(* Visualisation VISU_1_ENGINE
rectangle at (20,550)-(331,601): text "%s"; shows INPUTS.sVisuTime
rectangle at (15,0)-(326,51): text "ENGINE"
rectangle at (45,420)-(226,441): text "Coolant Temperature:%.0f ºC"; shows RECV_J1939.FEEE.EngineCoolantTemperature
rectangle at (45,440)-(226,461): text "Fuel Temperature:	%.0f ºC"; shows RECV_J1939.FEEE.EngineFuelTemperature
rounded rectangle at (900,50)-(1021,101): alarm colour if MAIN.aSys_Enable[8]
rounded rectangle at (905,55)-(1016,96): text "ENABLE / ENGINE"; alarm colour if MAIN.aSys_Enable[8]; taps MAIN.SIEngineEnable.In
rounded rectangle at (905,505)-(1016,546): text "RETURN"; opens VISU_0_MAIN
rounded rectangle at (905,395)-(1016,436): text "CONFIG: / ENGINE"; opens VISU_CFG_ENGINE
rounded rectangle at (905,450)-(1016,491): text "CONFIG: / PROPULSION"; opens VISU_CFG_PROPULSION
rectangle at (0,0)-(1,1): text "{ExtendedElement},Visu\ElementDLL.ete,0,@Zeigerinstrument,361,220,-40,1,0,0,128,1,RECV_J1939.F004.EngineActualSpeed,RPM,%.0f,0,0,0,200,600,0,3000,0,0,0,0,0,0,0,-24,180,700,MS Sans Serif,1,5,0,600,255,0,0,800,2400,0,255,0,2400,2800,255,255,0,2800,3000,255,0,0,600,800,255,255,0,0,255,255,255,,"
rectangle at (58,263)-(72,292): text "0"
rectangle at (12,135)-(54,164): text "600"
rectangle at (86,30)-(142,59): text "1200"
rectangle at (219,30)-(275,59): text "1800"
rectangle at (300,135)-(356,164): text "2400"
rectangle at (268,263)-(324,292): text "3000"
rectangle at (153,190)-(209,219): text "RPM"
polygon at (173,100)-(189,181): angle ((RECV_J1939.F004.EngineActualSpeed * 1.0)-1500) * 0.0866667
polygon at (178,82)-(183,94): angle ((RECV_J1939.F004.EngineActualSpeed * 1.0)-1500) * 0.0866667
rounded rectangle at (900,105)-(1021,156): alarm colour if MAIN.aSys_Enable[9]
rounded rectangle at (905,110)-(1016,151): text "ENABLE / PROPULSION"; alarm colour if MAIN.aSys_Enable[9]; taps MAIN.SIPropEnable.In
ellipse at (140,300)-(221,326): text "PROP."; alarm colour if ENGINE.Propulion_ON
ellipse at (135,245)-(226,276): text "%.0f"; shows RECV_J1939.F004.EngineActualSpeed
rectangle at (0,1)-(1,2): text "{ExtendedElement},Visu\ElementDLL.ete,1,@Bargraph,126,226,1,1,0,RECV_J1939.F004.EngineActualTorque,, %.0f,12.5,25,0,100,0,0,0,0,0,0,0,-20,150,700,MS Sans Serif,0,255,0,255,0,0,0,0,0,0,0,0,0,,1,"
rectangle at (21,113)-(47,211): alarm colour if (RECV_J1939.F004.EngineActualTorque) < 0; top ((RECV_J1939.F004.EngineActualTorque * 1.0) - 50)  * -1.96
rectangle at (48,194)-(117,227): text "0"
rectangle at (48,145)-(117,178): text "25"
rectangle at (48,97)-(117,130): text "50"
rectangle at (48,48)-(117,81): text "75"
rectangle at (48,0)-(117,32): text "100"
rectangle at (350,295)-(446,326): text "%d %%"; shows RECV_J1939.F004.EngineActualTorque
rectangle at (130,275)-(231,296): text "(Tgt= %.0f)"; shows ENGINE.fbEngine.Engine_RPM
rectangle at (645,415)-(716,436): text "%.1f bar"; shows P1101.Bar; alarm colour if P1101.Alarm.Adver; runs INTERN ASSIGN INPUTS.PresSelCalStbd[9]:=(FALSE)
rectangle at (645,435)-(716,456): text "%.1f bar"; shows P1102.Bar; alarm colour if P1102.Alarm.Adver; runs INTERN ASSIGN INPUTS.PresSelCalStbd[9]:=(FALSE)
rectangle at (245,420)-(426,441): text "Fuel Pressure:	%.1f MPa"; shows RECV_J1939.FEDB.EngineInjectorMeteringRail1Pressure
rectangle at (245,440)-(426,461): text "Engine Oil Pressure:	%.0f kPa"; shows RECV_J1939.FEEF.EngineOilPressure
rectangle at (245,460)-(426,481): text "Air Intake Pressure:	%.0f kPa"; shows RECV_J1939.FEF6.EngineIntakeMF1Pressure
rectangle at (245,480)-(426,501): text "Electrical Potential:	%.1f V"; shows RECV_J1939.FEF7.ElectricalPotential
rectangle at (135,365)-(226,386): text "%.0f RPM"; shows ENGINE.fbEngine.Forced_RPM; invisible if NOT PARAMS.stEngineCfg.EnForceRPM; runs INTERN ASSIGN INPUTS.PresSelCalStbd[9]:=(FALSE); editable
rectangle at (135,345)-(226,366): text "FORCED MIN"; shows RECV_J1939.F004.DriverDemandTorque; invisible if NOT PARAMS.stEngineCfg.EnForceRPM
ellipse at (40,330)-(111,401): invisible if NOT PARAMS.stEngineCfg.EnForceRPM; alarm colour if ENGINE.ForcedRPM
ellipse at (50,340)-(101,391): text "FORCE"; invisible if NOT PARAMS.stEngineCfg.EnForceRPM; toggles ENGINE.ForcedRPM
ellipse at (345,330)-(416,401): alarm colour if ENGINE.Engine_STOP
ellipse at (355,340)-(406,391): text "STOP"; taps ENGINE.Engine_STOP
rectangle at (775,350)-(856,371): text "%.0f bar"; shows P601.Bar; alarm colour if P601.Alarm.Adver; runs INTERN ASSIGN INPUTS.PresSelCalStbd[9]:=(FALSE)
rectangle at (775,430)-(856,451): text "%.1f %%"; shows LS601.Pos; alarm colour if LS601.Alarm.Adver; runs INTERN ASSIGN INPUTS.PresSelCalStbd[9]:=(FALSE)
rectangle at (0,0)-(1,1): text "{ExtendedElement},Visu\ElementDLL.ete,1,@Bargraph,86,21,3,0,0,LS601.Pos,,%,25,50,0,100,0,0,0,0,0,0,0,-13,16,700,Arial,0,255,0,255,0,0,0,0,0,0,0,0,0,,0,"
rectangle at (0,0)-(44,21): alarm colour if (LS601.Pos) < 0; right ((LS601.Pos * 1.0) - 50)  * 0.86
ellipse at (780,115)-(851,186): alarm colour if MAIN.fbDE601.OUT_EV3
ellipse at (780,205)-(851,276): alarm colour if MAIN.fbDE601.OUT_EV1
ellipse at (790,125)-(841,176): text "UP"; alarm colour if MAIN.fbDE601.IN_Hmi_CylIn; taps MAIN.fbDE601.IN_Hmi_CylIn
ellipse at (790,215)-(841,266): text "DW"; alarm colour if MAIN.fbDE601.IN_Hmi_CylOut; taps MAIN.fbDE601.IN_Hmi_CylOut
rectangle at (775,335)-(846,351): text "P601 - DW"
rectangle at (775,415)-(846,431): text "LS601"
ellipse at (775,485)-(816,506): text "UP"; alarm colour if MAIN.fbDE601.PROP_UP
ellipse at (815,485)-(856,506): text "DW"; alarm colour if MAIN.fbDE601.PROP_DW
rectangle at (775,390)-(856,411): text "%.0f bar"; shows P603.Bar; alarm colour if P603.Alarm.Adver; runs INTERN ASSIGN INPUTS.PresSelCalStbd[9]:=(FALSE)
rectangle at (775,375)-(846,391): text "P603 - UP"
rounded rectangle at (900,160)-(1021,211): alarm colour if MAIN.aHP_Enable[10]
rounded rectangle at (905,165)-(1016,206): text "ENABLE / PROP. UP/DW"; alarm colour if MAIN.aHP_Enable[10]; taps MAIN.SIPropUDEnable.In
rounded rectangle at (905,220)-(1016,261): text "MANUAL / PROP. UP"; alarm colour if MAIN.fbDE601.Man_Up; toggles MAIN.fbDE601.Man_Up
rounded rectangle at (905,275)-(1016,316): text "MANUAL / PROP. DW"; alarm colour if MAIN.fbDE601.Man_Dw; toggles MAIN.fbDE601.Man_Dw
rectangle at (45,500)-(226,521): text "Engine Fuel Rate:	%.1f L/h"; shows RECV_J1939.FEF2.EngineFuelRate
rectangle at (245,500)-(426,521): text "Total Hours:		%.1f hr"; shows RECV_J1939.FEE5.EngineTotalHoursOfOperation
rectangle at (45,480)-(226,501): text "Hydro Oil Temperature: %.0f ºC"; shows .S011.Deg; alarm colour if .S011.Alarm.Adver
rectangle at (190,55)-(286,81): text "ENGINE"
rectangle at (780,50)-(851,91): text "PROP. / UP/DW"
rectangle at (560,400)-(716,416): text "PROPULSION"; shows RECV_J1939.F004.DriverDemandTorque
rectangle at (570,75)-(631,106): text "FWD"
rectangle at (570,375)-(631,401): text "REV"
other_SCROLLBAR at (580,105)-(621,376): top ENGINE.ForcedProp_Thr; right PARAMS.stPropulsionCfg.aThrt_V[0]; bottom PARAMS.stPropulsionCfg.aThrt_V[10]
ellipse at (490,205)-(561,276): invisible if NOT PARAMS.stEngineCfg.EnForceTHR; alarm colour if ENGINE.ForcedProp
ellipse at (500,215)-(551,266): text "FORCE"; invisible if NOT PARAMS.stEngineCfg.EnForceTHR; toggles ENGINE.ForcedProp
ellipse at (640,205)-(711,276): alarm colour if ENGINE.ForcedProp_Thr = 0
ellipse at (650,215)-(701,266): text "IDLE"; runs INTERN ASSIGN ENGINE.ForcedProp_Thr:=(0)
rectangle at (485,415)-(556,436): text "%.2f V"; shows ENGINE.fbPropulsion.Throttle_V; alarm colour if ENGINE.fbPropulsion.Throttle_err; runs INTERN ASSIGN INPUTS.PresSelCalStbd[9]:=(FALSE)
rectangle at (485,435)-(556,456): text "%.0f rpm"; shows ENGINE.fbPropulsion.Tgt_RPM; runs INTERN ASSIGN INPUTS.PresSelCalStbd[9]:=(FALSE)
rectangle at (560,435)-(646,456): text "REV: %d mA"; shows ENGINE.fbPropulsion.RevEVP; runs INTERN ASSIGN INPUTS.PresSelCalStbd[9]:=(FALSE)
rectangle at (560,415)-(646,436): text "FWD: %d mA"; shows ENGINE.fbPropulsion.FwdEVP; runs INTERN ASSIGN INPUTS.PresSelCalStbd[9]:=(FALSE)
rectangle at (485,400)-(556,416): text "THROTTLE"; shows RECV_J1939.F004.DriverDemandTorque
rectangle at (540,55)-(661,81): text "THROTTLE"
rectangle at (550,505)-(656,526): text "EVP001: %d mA"; shows EVP001; alarm colour if EVP001 = 0
rectangle at (550,485)-(656,506): text "EVP002: %d mA"; shows EVP002; alarm colour if EVP002 = 0
ellipse at (660,495)-(711,516): text "EV1101"; alarm colour if EV1101
rounded rectangle at (905,335)-(1016,376): text "CLEAR"; alarm colour if ALARMS.Clear; taps ALARMS.Clear
rectangle at (550,460)-(656,481): text "S1100: %.0f °C"; shows S1100.Deg; alarm colour if S1100.Alarm.Adver
rounded rectangle at (660,460)-(711,481): text "MUTE"; alarm colour if ENGINE.S1100_Mute; toggles ENGINE.S1100_Mute
rectangle at (485,460)-(551,481): text "Temp"; shows RECV_J1939.F004.DriverDemandTorque
rectangle at (45,460)-(226,481): text "Exaust Temperature: %.0f ºC"; shows S100.Deg; alarm colour if S100.Alarm.Adver
41 more shapes without text or variables
*)

(* Visualisation VISU_1_KEEL
rectangle at (20,550)-(331,601): text "%s"; shows INPUTS.sVisuTime
rounded rectangle at (905,505)-(1016,546): text "RETURN"; opens VISU_0_MAIN
rectangle at (15,0)-(581,51): text "KEEL && DAGGERBOARD"
rectangle at (185,390)-(286,411): text "P1001: %.0f bar"; shows P1001.Bar; alarm colour if P1001.Alarm.Adver; runs INTERN ASSIGN INPUTS.PresSelCalStbd[9]:=(FALSE)
rectangle at (115,420)-(216,441): text "LS1001: %.1f %%"; shows LS1001.Pos; alarm colour if LS1001.Alarm.Adver; runs INTERN ASSIGN INPUTS.PresSelCalStbd[9]:=(FALSE)
rectangle at (0,0)-(1,1): text "{ExtendedElement},Visu\ElementDLL.ete,1,@Bargraph,61,11,3,0,1,LS1001.Pos,,%,25,50,50,100,0,0,0,0,0,0,0,-13,16,700,Arial,0,255,0,255,0,0,1,50,0,0,0,0,0,,0,"
rectangle at (31,0)-(62,11): alarm colour if (LS1001.Pos) > 50; left ((LS1001.Pos * 1.0) - 75)  * -1.2
ellipse at (40,160)-(111,231): alarm colour if MAIN.fbKeel.MOVING_O
ellipse at (220,160)-(291,231): alarm colour if MAIN.fbKeel.MOVING_I
ellipse at (50,170)-(101,221): text "PORT"; alarm colour if MAIN.fbKeel.IN_Hmi_O; taps MAIN.fbKeel.IN_Hmi_O
ellipse at (230,170)-(281,221): text "STBD"; alarm colour if MAIN.fbKeel.IN_Hmi_I; taps MAIN.fbKeel.IN_Hmi_I
rectangle at (145,55)-(196,86): text "KEEL"
ellipse at (190,490)-(231,511): text "STBD"; alarm colour if MAIN.fbKeel.KEEL_I
ellipse at (100,490)-(141,511): text "PORT"; alarm colour if MAIN.fbKeel.KEEL_O
rounded rectangle at (40,95)-(111,131): text "ENABLE"; alarm colour if MAIN.aLP_Enable[13]; toggles MAIN.aLP_Enable[13]
rectangle at (45,390)-(146,411): text "P1002: %.0f bar"; shows P1002.Bar; alarm colour if P1002.Alarm.Adver; runs INTERN ASSIGN INPUTS.PresSelCalStbd[9]:=(FALSE)
ellipse at (145,490)-(186,511): text "CENT"; alarm colour if MAIN.fbKeel.KEEL_C
rounded rectangle at (905,115)-(1016,156): text "MANUAL / KEEL"; alarm colour if MAIN.fbKEEL.Manual; toggles MAIN.fbKEEL.Manual
ellipse at (130,160)-(201,231): alarm colour if MAIN.fbKeel.MOVING_F
ellipse at (140,170)-(191,221): text "FLOAT"; alarm colour if MAIN.fbKeel.IN_Hmi_F; taps MAIN.fbKeel.IN_Hmi_F
ellipse at (135,100)-(206,126): text "ENGINE"; alarm colour if MAIN.fbKEEL.EngReady
ellipse at (635,160)-(706,231): invisible if MAIN.fbBoard.Manual = FALSE; alarm colour if MAIN.fbBoard.MOVING_P_In
ellipse at (635,250)-(706,321): invisible if MAIN.fbBoard.Manual = FALSE; alarm colour if MAIN.fbBoard.MOVING_P_Out
ellipse at (645,170)-(696,221): text "PUMP"; invisible if MAIN.fbBoard.Manual = FALSE; alarm colour if MAIN.fbBoard.IN_Hmi_P_In; taps MAIN.fbBoard.IN_Hmi_P_In
ellipse at (645,260)-(696,311): text "EASE"; invisible if MAIN.fbBoard.Manual = FALSE; alarm colour if MAIN.fbBoard.IN_Hmi_P_Out; taps MAIN.fbBoard.IN_Hmi_P_Out
rectangle at (635,55)-(706,86): text "DGBD / PORT"
rounded rectangle at (605,95)-(676,131): text "ENABLE"; alarm colour if MAIN.aLP_Enable[11]; toggles MAIN.aLP_Enable[11]
ellipse at (755,160)-(826,231): invisible if MAIN.fbBoard.Manual = FALSE; alarm colour if MAIN.fbBoard.MOVING_S_In
ellipse at (755,250)-(826,321): invisible if MAIN.fbBoard.Manual = FALSE; alarm colour if MAIN.fbBoard.MOVING_S_Out
ellipse at (765,170)-(816,221): text "PUMP"; invisible if MAIN.fbBoard.Manual = FALSE; alarm colour if MAIN.fbBoard.IN_Hmi_S_In; taps MAIN.fbBoard.IN_Hmi_S_In
ellipse at (765,260)-(816,311): text "EASE"; invisible if MAIN.fbBoard.Manual = FALSE; alarm colour if MAIN.fbBoard.IN_Hmi_S_Out; taps MAIN.fbBoard.IN_Hmi_S_Out
rectangle at (755,55)-(826,86): text "DGBD / STBD"
rectangle at (610,420)-(711,441): text "LS801: %.1f %%"; shows LS801.Pos; alarm colour if LS801.Alarm.Adver; runs INTERN ASSIGN INPUTS.PresSelCalStbd[9]:=(FALSE)
rectangle at (0,0)-(1,1): text "{ExtendedElement},Visu\ElementDLL.ete,1,@Bargraph,106,21,3,0,0,LS801.Pos,,%,25,50,0,100,0,0,0,0,0,0,0,-13,16,700,Arial,0,255,0,255,0,0,0,0,0,0,0,0,0,,0,"
rectangle at (0,0)-(54,21): alarm colour if (LS801.Pos) < 0; right ((LS801.Pos * 1.0) - 50)  * 1.06
rectangle at (750,420)-(851,441): text "LS803: %.1f %%"; shows LS803.Pos; alarm colour if LS803.Alarm.Adver; runs INTERN ASSIGN INPUTS.PresSelCalStbd[9]:=(FALSE)
rectangle at (0,0)-(1,1): text "{ExtendedElement},Visu\ElementDLL.ete,1,@Bargraph,106,21,3,0,1,LS803.Pos,,%,25,50,0,100,0,0,0,0,0,0,0,-13,16,700,Arial,0,255,0,255,0,0,0,0,0,0,0,0,0,,0,"
rectangle at (53,0)-(107,21): alarm colour if (LS803.Pos) < 0; left ((LS803.Pos * 1.0) - 50)  * -1.06
rectangle at (610,370)-(711,391): text "P802: %.0f bar"; shows P802.Bar; alarm colour if P802.Alarm.Adver; runs INTERN ASSIGN INPUTS.PresSelCalStbd[9]:=(FALSE)
rectangle at (610,390)-(711,411): text "P1216: %.0f bar"; shows P1216.Bar; alarm colour if P1216.Alarm.Adver; runs INTERN ASSIGN INPUTS.PresSelCalStbd[9]:=(FALSE)
rectangle at (750,370)-(851,391): text "P804: %.0f bar"; shows P804.Bar; alarm colour if P804.Alarm.Adver; runs INTERN ASSIGN INPUTS.PresSelCalStbd[9]:=(FALSE)
rectangle at (750,390)-(851,411): text "P1219: %.0f bar"; shows P1219.Bar; alarm colour if P1219.Alarm.Adver; runs INTERN ASSIGN INPUTS.PresSelCalStbd[9]:=(FALSE)
ellipse at (595,500)-(636,521): text "SF801"; alarm colour if SF801.Alarm.Alarm
ellipse at (735,500)-(776,521): text "SF803"; alarm colour if SF803.Alarm.Alarm
rectangle at (115,450)-(216,471): text "LS1002: %.1f %%"; shows LS1002.Pos; alarm colour if LS1002.Alarm.Adver; runs INTERN ASSIGN INPUTS.PresSelCalStbd[9]:=(FALSE)
rectangle at (0,0)-(1,1): text "{ExtendedElement},Visu\ElementDLL.ete,1,@Bargraph,61,11,3,0,1,LS1002.Pos,,%,25,50,50,100,0,0,0,0,0,0,0,-13,16,700,Arial,0,255,0,255,0,0,1,50,0,0,0,0,0,,0,"
rectangle at (31,0)-(62,11): alarm colour if (LS1002.Pos) > 50; left ((LS1002.Pos * 1.0) - 75)  * -1.2
ellipse at (230,100)-(281,126): text "SF1002"; alarm colour if SF1002.Alarm.Alarm
rounded rectangle at (905,170)-(1016,211): text "MANUAL / BOARD"; alarm colour if MAIN.fbBoard.Manual; toggles MAIN.fbBoard.Manual
ellipse at (590,205)-(661,276): invisible if MAIN.fbBoard.Manual; alarm colour if MAIN.fbBoard.MOVING_P
ellipse at (800,205)-(871,276): invisible if MAIN.fbBoard.Manual; alarm colour if MAIN.fbBoard.MOVING_S
ellipse at (600,215)-(651,266): text "PORT"; invisible if MAIN.fbBoard.Manual; alarm colour if MAIN.fbBoard.IN_Hmi_P; taps MAIN.fbBoard.IN_Hmi_P
ellipse at (810,215)-(861,266): text "STBD"; invisible if MAIN.fbBoard.Manual; alarm colour if MAIN.fbBoard.IN_Hmi_S; taps MAIN.fbBoard.IN_Hmi_S
ellipse at (695,205)-(766,276): invisible if MAIN.fbBoard.Manual; alarm colour if MAIN.fbBoard.MOVING_C
ellipse at (705,215)-(756,266): text "CENTER"; invisible if MAIN.fbBoard.Manual; alarm colour if MAIN.fbBoard.IN_Hmi_C; taps MAIN.fbBoard.IN_Hmi_C
ellipse at (700,100)-(771,126): text "ENGINE"; alarm colour if MAIN.fbBoard.EngReady
rounded rectangle at (710,270)-(751,301): text "%d %%"; shows MAIN.fbBoard.IN_Hmi_OutPerc; invisible if MAIN.fbBoard.Manual = FALSE; editable 5..100
rounded rectangle at (710,180)-(751,211): text "%d %%"; shows MAIN.fbBoard.IN_Hmi_InPerc; invisible if MAIN.fbBoard.Manual = FALSE; editable 5..100
rectangle at (610,340)-(711,361): text "EVP1216: %d %%"; shows EVP1216_7 / 10; alarm colour if EVP1216_7 = 0
rectangle at (750,340)-(851,361): text "EVP1218: %d %%"; shows EVP1218_9 / 10; alarm colour if EVP1218_9 = 0
rectangle at (45,340)-(146,361): text "EVP1220: %d %%"; shows EVP1220_1 / 10; alarm colour if EVP1220_1 = 0
ellipse at (595,470)-(636,491): text "PORT"; alarm colour if MAIN.fbBoard.LS_P_Out
ellipse at (640,470)-(681,491): text "CENT"; alarm colour if MAIN.fbBoard.LS_P_Mid
ellipse at (735,470)-(776,491): text "PORT"; alarm colour if MAIN.fbBoard.LS_S_In
ellipse at (825,470)-(866,491): text "STBD"; alarm colour if MAIN.fbBoard.LS_S_Out
ellipse at (780,470)-(821,491): text "CENT"; alarm colour if MAIN.fbBoard.LS_S_Mid
ellipse at (130,250)-(201,321): alarm colour if MAIN.fbKeel.MOVING_C
ellipse at (140,260)-(191,311): text "CENTER"; alarm colour if MAIN.fbKeel.IN_Hmi_C; taps MAIN.fbKeel.IN_Hmi_C
ellipse at (220,250)-(291,321): alarm colour if MAIN.fbKeel.MOVING_T
ellipse at (230,260)-(281,311): text "TACK"; alarm colour if MAIN.fbKeel.IN_Hmi_T; taps MAIN.fbKeel.IN_Hmi_T
ellipse at (135,505)-(151,521): text "S"; alarm colour if MAIN.fbKeel.KEEL_SO
ellipse at (180,505)-(196,521): text "S"; alarm colour if MAIN.fbKeel.KEEL_SI
ellipse at (685,470)-(726,491): text "STBD"; alarm colour if MAIN.fbBoard.LS_P_In
ellipse at (815,485)-(831,501): text "S"; alarm colour if MAIN.fbBoard.LS_Safe_S_Out
ellipse at (770,485)-(786,501): text "S"; alarm colour if MAIN.fbBoard.LS_Safe_S_In
ellipse at (675,485)-(691,501): text "S"; alarm colour if MAIN.fbBoard.LS_Safe_P_In
ellipse at (630,485)-(646,501): text "S"; alarm colour if MAIN.fbBoard.LS_Safe_P_Out
rectangle at (45,360)-(146,381): text "EVP002: %d mA"; shows EVP002; alarm colour if EVP002 = 0
rectangle at (185,360)-(286,381): text "EVP001: %d mA"; shows EVP001; alarm colour if EVP001 = 0
rounded rectangle at (905,395)-(1016,436): text "KEEL"; opens VISU_2_KEEL
rounded rectangle at (905,450)-(1016,491): text "BOARD"; opens VISU_2_BOARD
ellipse at (240,425)-(291,451): text "SF1003"; alarm colour if SF1003.Alarm.Alarm
ellipse at (240,455)-(291,481): text "SF1004"; alarm colour if SF1004.Alarm.Alarm
rounded rectangle at (905,55)-(1016,96): text "CLEAR"; alarm colour if ALARMS.Clear; taps ALARMS.Clear
14 more shapes without text or variables
*)

(* Visualisation VISU_1_PUMPS
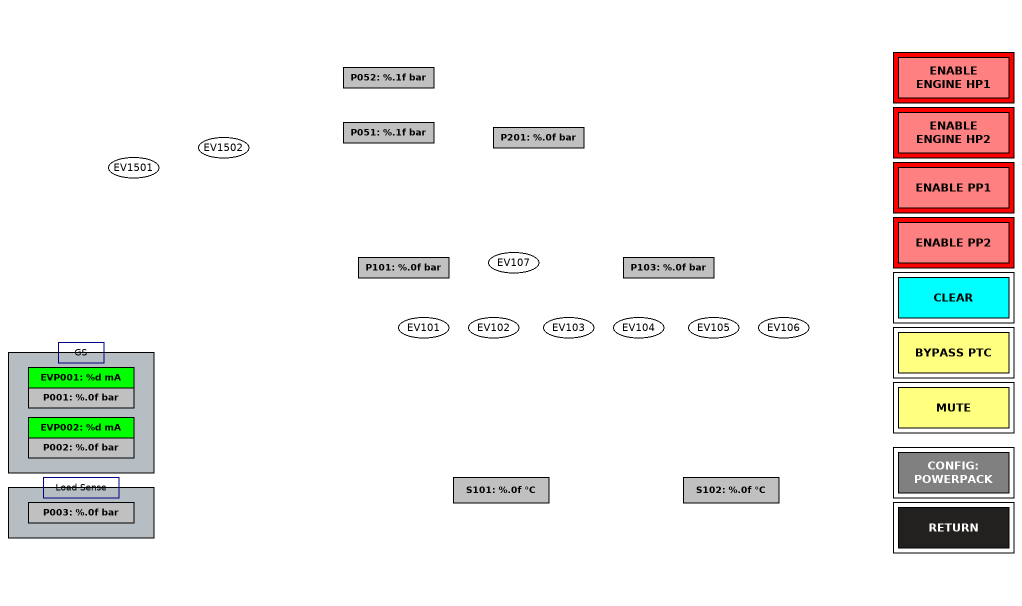
rectangle at (65,340)-(111,361): text "GS"
rectangle at (20,0)-(331,51): text "PUMPS"
rectangle at (20,550)-(331,601): text "%s"; shows INPUTS.sVisuTime
rounded rectangle at (905,505)-(1016,546): text "RETURN"; opens VISU_0_MAIN
rectangle at (35,385)-(141,406): text "P001: %.0f bar"; shows P001.Bar; alarm colour if P001.Alarm.Adver
rectangle at (35,435)-(141,456): text "P002: %.0f bar"; shows P002.Bar; alarm colour if P002.Alarm.Adver
ellipse at (765,315)-(816,336): text "EV106"; alarm colour if EV106
ellipse at (695,315)-(746,336): text "EV105"; alarm colour if EV105
rounded rectangle at (900,160)-(1021,211): alarm colour if MAIN.aSys_Enable[6]
rounded rectangle at (905,165)-(1016,206): text "ENABLE PP1"; alarm colour if MAIN.aSys_Enable[6]; toggles MAIN.aSys_Enable[6]
rounded rectangle at (900,215)-(1021,266): alarm colour if MAIN.aSys_Enable[7]
rounded rectangle at (905,220)-(1016,261): text "ENABLE PP2"; alarm colour if MAIN.aSys_Enable[7]; toggles MAIN.aSys_Enable[7]
rounded rectangle at (905,450)-(1016,491): text "CONFIG: / POWERPACK"; opens VISU_CFG_POWERPACK
rounded rectangle at (905,330)-(1016,371): text "BYPASS PTC"; alarm colour if POWERPACK.Bypass; toggles POWERPACK.Bypass
rounded rectangle at (905,385)-(1016,426): text "MUTE"; alarm colour if POWERPACK.Mute; toggles POWERPACK.Mute
rectangle at (35,365)-(141,386): text "EVP001: %d mA"; shows EVP001; alarm colour if EVP001 = 0
rounded rectangle at (900,50)-(1021,101): alarm colour if MAIN.aSys_Enable[4]
rounded rectangle at (905,55)-(1016,96): text "ENABLE / ENGINE HP1"; alarm colour if MAIN.aSys_Enable[4]; toggles MAIN.aSys_Enable[4]
rounded rectangle at (900,105)-(1021,156): alarm colour if MAIN.aSys_Enable[5]
rounded rectangle at (905,110)-(1016,151): text "ENABLE / ENGINE HP2"; alarm colour if MAIN.aSys_Enable[5]; toggles MAIN.aSys_Enable[5]
rectangle at (35,415)-(141,436): text "EVP002: %d mA"; shows EVP002; alarm colour if EVP002 = 0
rectangle at (350,120)-(441,141): text "P051: %.1f bar"; shows P051.Bar; alarm colour if P051.Alarm.Adver
rectangle at (350,65)-(441,86): text "P052: %.1f bar"; shows P052.Bar; alarm colour if P052.Alarm.Adver
rectangle at (365,255)-(456,276): text "P101: %.0f bar"; shows P101.Bar; alarm colour if P101.Alarm.Adver
rectangle at (630,255)-(721,276): text "P103: %.0f bar"; shows P103.Bar; alarm colour if P103.Alarm.Adver
ellipse at (620,315)-(671,336): text "EV104"; alarm colour if EV104
ellipse at (550,315)-(601,336): text "EV103"; alarm colour if EV103
ellipse at (475,315)-(526,336): text "EV102"; alarm colour if EV102
ellipse at (405,315)-(456,336): text "EV101"; alarm colour if EV101
ellipse at (495,250)-(546,271): text "EV107"; alarm colour if EV107
ellipse at (205,135)-(256,156): text "EV1502"; alarm colour if EV1502
ellipse at (115,155)-(166,176): text "EV1501"; alarm colour if EV1501
rectangle at (500,125)-(591,146): text "P201: %.0f bar"; shows P201.Bar; alarm colour if P201.Alarm.Adver
rounded rectangle at (905,275)-(1016,316): text "CLEAR"; alarm colour if ALARMS.Clear; taps ALARMS.Clear
rectangle at (690,475)-(786,501): text "S102: %.0f °C"; shows S102.Deg; alarm colour if S102.Alarm.Adver
rectangle at (460,475)-(556,501): text "S101: %.0f °C"; shows S101.Deg; alarm colour if S101.Alarm.Adver
rectangle at (50,475)-(126,496): text "Load Sense"
rectangle at (35,500)-(141,521): text "P003: %.0f bar"; shows P003.Bar; alarm colour if P003.Alarm.Adver
7 more shapes without text or variables
*)

(* Visualisation VISU_1_SPECIAL
rectangle at (20,550)-(331,601): text "%s"; shows INPUTS.sVisuTime
rounded rectangle at (905,505)-(1016,546): text "RETURN"; opens VISU_0_MAIN
rectangle at (20,0)-(331,51): text "SPECIAL"
rectangle at (180,380)-(281,401): text "P605: %.0f bar"; shows P605.Bar; alarm colour if P605.Alarm.Adver; runs INTERN ASSIGN INPUTS.PresSelCalStbd[9]:=(FALSE)
rectangle at (180,430)-(281,451): text "LS605: %.1f %%"; shows LS605.Pos; alarm colour if LS605.Alarm.Adver; runs INTERN ASSIGN INPUTS.PresSelCalStbd[9]:=(FALSE)
rectangle at (0,0)-(1,1): text "{ExtendedElement},Visu\ElementDLL.ete,1,@Bargraph,86,21,3,0,0,LS605.Pos,,%,25,50,0,100,0,0,0,0,0,0,0,-13,16,700,Arial,0,255,0,255,0,0,0,0,0,0,0,0,0,,0,"
rectangle at (0,0)-(44,21): alarm colour if (LS605.Pos) < 0; right ((LS605.Pos * 1.0) - 50)  * 0.86
ellipse at (160,165)-(231,236): alarm colour if MAIN.fbDE605.OUT_EV3
ellipse at (160,245)-(231,316): alarm colour if MAIN.fbDE605.OUT_EV1
ellipse at (170,175)-(221,226): text "PORT"; alarm colour if MAIN.fbDE605.IN_Hmi_CylIn; taps MAIN.fbDE605.IN_Hmi_CylIn
ellipse at (170,255)-(221,306): text "STBD"; alarm colour if MAIN.fbDE605.IN_Hmi_CylOut; taps MAIN.fbDE605.IN_Hmi_CylOut
rectangle at (205,55)-(256,86): text "TRIM / TAB"
ellipse at (190,480)-(231,501): text "IN"; alarm colour if MAIN.fbDE605.LS_In
ellipse at (230,480)-(271,501): text "OUT"; alarm colour if MAIN.fbDE605.LS_Out
rounded rectangle at (195,100)-(266,136): text "ENABLE"; alarm colour if MAIN.aHP_Enable[11]; toggles MAIN.aHP_Enable[11]
rectangle at (180,400)-(281,421): text "P607: %.0f bar"; shows P607.Bar; alarm colour if P607.Alarm.Adver; runs INTERN ASSIGN INPUTS.PresSelCalStbd[9]:=(FALSE)
ellipse at (210,500)-(251,521): text "CENT"; alarm colour if MAIN.fbDE605.LS_Mid
rectangle at (25,380)-(126,401): text "P601Dw: %.0f bar"; shows P601.Bar; alarm colour if P601.Alarm.Adver; runs INTERN ASSIGN INPUTS.PresSelCalStbd[9]:=(FALSE)
rectangle at (25,430)-(126,451): text "LS601: %.1f %%"; shows LS601.Pos; alarm colour if LS601.Alarm.Adver; runs INTERN ASSIGN INPUTS.PresSelCalStbd[9]:=(FALSE)
rectangle at (0,0)-(1,1): text "{ExtendedElement},Visu\ElementDLL.ete,1,@Bargraph,106,21,3,0,0,LS601.Pos,,%,25,50,0,100,0,0,0,0,0,0,0,-13,16,700,Arial,0,255,0,255,0,0,0,0,0,0,0,0,0,,0,"
rectangle at (0,0)-(54,21): alarm colour if (LS601.Pos) < 0; right ((LS601.Pos * 1.0) - 50)  * 1.06
ellipse at (40,165)-(111,236): alarm colour if MAIN.fbDE601.OUT_EV3
ellipse at (40,245)-(111,316): alarm colour if MAIN.fbDE601.OUT_EV1
ellipse at (50,175)-(101,226): text "UP"; alarm colour if MAIN.fbDE601.IN_Hmi_CylIn; taps MAIN.fbDE601.IN_Hmi_CylIn
ellipse at (50,255)-(101,306): text "DW"; alarm colour if MAIN.fbDE601.IN_Hmi_CylOut; taps MAIN.fbDE601.IN_Hmi_CylOut
rectangle at (50,55)-(101,86): text "PROP. / UP/DW"
ellipse at (35,480)-(76,501): text "UP"; alarm colour if MAIN.fbDE601.PROP_UP
ellipse at (75,480)-(116,501): text "DW"; alarm colour if MAIN.fbDE601.PROP_DW
rounded rectangle at (40,100)-(111,136): text "ENABLE"; alarm colour if MAIN.aHP_Enable[10]; toggles MAIN.aHP_Enable[10]
rectangle at (25,400)-(126,421): text "P603Up: %.0f bar"; shows P603.Bar; alarm colour if P603.Alarm.Adver; runs INTERN ASSIGN INPUTS.PresSelCalStbd[9]:=(FALSE)
rounded rectangle at (905,245)-(1016,286): text "MANUAL / PROP. UP"; alarm colour if MAIN.fbDE601.Man_Up; toggles MAIN.fbDE601.Man_Up
rounded rectangle at (905,300)-(1016,341): text "MANUAL / PROP. DW"; alarm colour if MAIN.fbDE601.Man_Dw; toggles MAIN.fbDE601.Man_Dw
rounded rectangle at (905,450)-(1016,491): text "CONFIG: / SPECIAL"; opens VISU_CFG_SPECIAL
rounded rectangle at (905,395)-(1016,436): text "CALIB: / SPECIAL"; opens VISU_CAL_SPECIAL
rectangle at (370,380)-(471,401): text "P1301: %.0f bar"; shows P1301.Bar; alarm colour if P1301.Alarm.Adver; runs INTERN ASSIGN INPUTS.PresSelCalStbd[9]:=(FALSE)
rectangle at (370,430)-(471,451): text "LS1303: %.1f %%"; shows LS1303.Pos; alarm colour if LS1303.Alarm.Adver; runs INTERN ASSIGN INPUTS.PresSelCalStbd[9]:=(FALSE)
rectangle at (0,0)-(1,1): text "{ExtendedElement},Visu\ElementDLL.ete,1,@Bargraph,56,21,3,0,1,LS1303.Pos,,%,25,50,50,100,0,0,0,0,0,0,0,-13,16,700,Arial,0,255,0,255,0,0,1,50,0,0,0,0,0,,0,"
rectangle at (28,0)-(57,21): alarm colour if (LS1303.Pos) > 50; left ((LS1303.Pos * 1.0) - 75)  * -1.12
ellipse at (350,165)-(421,236): alarm colour if MAIN.fbTraveller.Move_B
ellipse at (350,245)-(421,316): alarm colour if MAIN.fbTraveller.Move_A
ellipse at (360,175)-(411,226): text "PORT"; alarm colour if MAIN.fbTraveller.IN_Hmi_B; taps MAIN.fbTraveller.IN_Hmi_B
ellipse at (360,255)-(411,306): text "STBD"; alarm colour if MAIN.fbTraveller.IN_Hmi_A; taps MAIN.fbTraveller.IN_Hmi_A
rectangle at (385,55)-(456,86): text "TRAVELLER"
ellipse at (380,480)-(421,501): text "PORT"; alarm colour if MAIN.fbTraveller.LS_Max
ellipse at (420,480)-(461,501): text "STBD"; alarm colour if MAIN.fbTraveller.LS_Min
rounded rectangle at (385,100)-(456,136): text "ENABLE"; alarm colour if MAIN.aLP_Enable[16]; toggles MAIN.aLP_Enable[16]
rectangle at (370,400)-(471,421): text "P1302: %.0f bar"; shows P1302.Bar; alarm colour if P1302.Alarm.Adver; runs INTERN ASSIGN INPUTS.PresSelCalStbd[9]:=(FALSE)
ellipse at (400,500)-(441,521): text "CENT"; alarm colour if MAIN.fbTraveller.LS_Mid
rectangle at (540,55)-(611,86): text "BOW / THR"
rounded rectangle at (540,100)-(611,136): text "ENABLE"; alarm colour if MAIN.aLP_Enable[17]; toggles MAIN.aLP_Enable[17]
rectangle at (660,55)-(731,86): text "BOW THR / UP/DW"
rounded rectangle at (660,100)-(731,136): text "ENABLE"; alarm colour if MAIN.aLP_Enable[18]; toggles MAIN.aLP_Enable[18]
ellipse at (540,165)-(611,236): alarm colour if MAIN.fbBowThr.OUT_1
ellipse at (540,245)-(611,316): alarm colour if MAIN.fbBowThr.OUT_2
ellipse at (550,175)-(601,226): text "1 P"; alarm colour if MAIN.fbBowThr.IN_Hmi_1; taps MAIN.fbBowThr.IN_Hmi_1
ellipse at (550,255)-(601,306): text "2 S"; alarm colour if MAIN.fbBowThr.IN_Hmi_2; taps MAIN.fbBowThr.IN_Hmi_2
ellipse at (660,165)-(731,236): alarm colour if MAIN.fbBowThrUpDw.OUT_1
ellipse at (660,245)-(731,316): alarm colour if MAIN.fbBowThrUpDw.OUT_2
ellipse at (670,175)-(721,226): text "1 UP"; alarm colour if MAIN.fbBowThrUpDw.IN_Hmi_1; taps MAIN.fbBowThrUpDw.IN_Hmi_1
ellipse at (670,255)-(721,306): text "2 DW"; alarm colour if MAIN.fbBowThrUpDw.IN_Hmi_2; taps MAIN.fbBowThrUpDw.IN_Hmi_2
rectangle at (525,350)-(626,371): text "EVP402: %d %%"; shows EVP402_3 / 10; alarm colour if EVP402_3 = 0
rectangle at (645,350)-(746,371): text "EVP404: %d %%"; shows EVP404_5 / 10; alarm colour if EVP404_5 = 0
ellipse at (675,385)-(716,406): text "UP"; alarm colour if MAIN.fbBowThrUpDw.IN_SF1
ellipse at (675,405)-(716,426): text "DW"; alarm colour if MAIN.fbBowThrUpDw.IN_SF2
rectangle at (370,350)-(471,371): text "EVP1606: %d %%"; shows EVP1606_7 / 10; alarm colour if EVP1606_7 = 0
ellipse at (240,215)-(291,266): text "CENTER"; alarm colour if MAIN.fbDE605.IN_Hmi_CylMid; taps MAIN.fbDE605.IN_Hmi_CylMid
ellipse at (430,215)-(481,266): text "TACK"; alarm colour if MAIN.fbTraveller.IN_Hmi_T; taps MAIN.fbTraveller.IN_Hmi_T
rounded rectangle at (905,55)-(1016,96): text "CLEAR"; alarm colour if ALARMS.Clear; taps ALARMS.Clear
rectangle at (780,55)-(851,86): text "TACK / VALVE"
rounded rectangle at (785,100)-(856,136): text "ENABLE"; alarm colour if MAIN.aSys_Enable[16]; toggles MAIN.aSys_Enable[16]
ellipse at (770,235)-(836,301): alarm colour if MAIN.fbTackValve.Port_Close
ellipse at (780,245)-(826,291): text "CLOSE"; alarm colour if MAIN.fbTackValve.OUT_Port_Close; taps MAIN.fbTackValve.IN_Hmi_Port_Close
ellipse at (770,160)-(836,226): alarm colour if MAIN.fbTackValve.Port_Open
ellipse at (780,170)-(826,216): text "OPEN"; alarm colour if MAIN.fbTackValve.OUT_Port_Open; taps MAIN.fbTackValve.IN_Hmi_Port_Open
ellipse at (805,370)-(871,436): alarm colour if MAIN.fbTackValve.Stbd_Close
ellipse at (815,380)-(861,426): text "CLOSE"; alarm colour if MAIN.fbTackValve.OUT_Stbd_Close; taps MAIN.fbTackValve.IN_Hmi_Stbd_Close
ellipse at (805,445)-(871,511): alarm colour if MAIN.fbTackValve.Stbd_Open
ellipse at (815,455)-(861,501): text "OPEN"; alarm colour if MAIN.fbTackValve.OUT_Stbd_Open; taps MAIN.fbTackValve.IN_Hmi_Stbd_Open
rectangle at (770,315)-(871,336): text "Heel: %.1f º"; shows TOFARO.rHeel; alarm colour if TOFARO.Recv_Live; runs INTERN ASSIGN INPUTS.PresSelCalStbd[9]:=(FALSE)
rectangle at (0,0)-(1,1): text "{ExtendedElement},Visu\ElementDLL.ete,1,@Bargraph,56,21,3,0,0,TOFARO.rHeel,,%,5,25,0,50,0,0,0,0,0,0,0,-13,16,700,Arial,0,255,0,255,0,0,0,0,0,0,0,0,0,,0,"
rectangle at (0,0)-(29,21): alarm colour if (TOFARO.rHeel) < 0; right ((TOFARO.rHeel * 1.0) - 25)  * 1.12
rounded rectangle at (900,145)-(1021,196): alarm colour if MAIN.fbTackValve.Manual
rounded rectangle at (905,150)-(1016,191): text "MANUAL / TACK VALVE"; alarm colour if MAIN.fbTackValve.Manual; toggles MAIN.fbTackValve.Manual
ellipse at (830,220)-(871,241): text "RDY"; alarm colour if MAIN.fbTackValve.Port_Ready
ellipse at (770,430)-(811,451): text "RDY"; alarm colour if MAIN.fbTackValve.Stbd_Ready
24 more shapes without text or variables
*)

(* Visualisation VISU_1_TANK
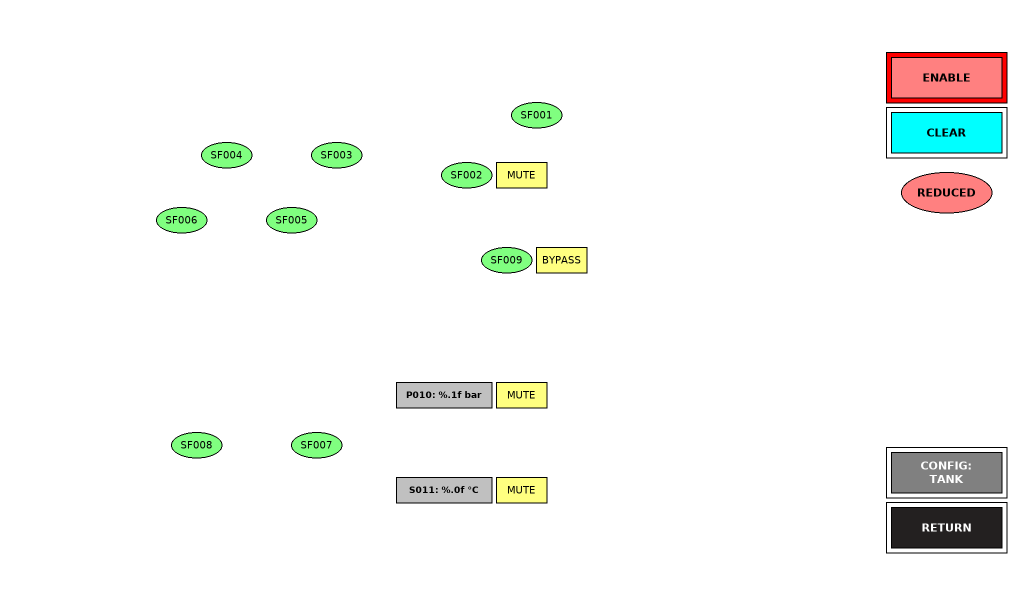
rectangle at (20,0)-(331,51): text "TANK"
rectangle at (410,380)-(506,406): text "P010: %.1f bar"; shows P010.Bar; alarm colour if P010.Alarm.Adver
ellipse at (215,140)-(266,166): text "SF004"; alarm colour if SF004.Alarm.Adver
ellipse at (455,160)-(506,186): text "SF002"; alarm colour if SF002.Alarm.Adver
rounded rectangle at (510,160)-(561,186): text "MUTE"; alarm colour if TANK.SF002_Mute; toggles TANK.SF002_Mute
rounded rectangle at (510,380)-(561,406): text "MUTE"; alarm colour if TANK.P010_Mute; toggles TANK.P010_Mute
rounded rectangle at (905,505)-(1016,546): text "RETURN"; opens VISU_0_MAIN
rectangle at (20,550)-(331,601): text "%s"; shows INPUTS.sVisuTime
rounded rectangle at (900,50)-(1021,101): alarm colour if MAIN.aSys_Enable[1]
rounded rectangle at (905,55)-(1016,96): text "ENABLE"; alarm colour if MAIN.aSys_Enable[1]; taps MAIN.SITankEnable.In
rounded rectangle at (905,450)-(1016,491): text "CONFIG: / TANK"; opens VISU_CFG_TANK
ellipse at (170,205)-(221,231): text "SF006"; alarm colour if SF006.Alarm.Adver
ellipse at (185,430)-(236,456): text "SF008"; alarm colour if SF008.Alarm.Adver
ellipse at (325,140)-(376,166): text "SF003"; alarm colour if SF003.Alarm.Adver
ellipse at (280,205)-(331,231): text "SF005"; alarm colour if SF005.Alarm.Adver
ellipse at (305,430)-(356,456): text "SF007"; alarm colour if SF007.Alarm.Adver
ellipse at (525,100)-(576,126): text "SF001"; alarm colour if SF001.Alarm.Adver
rectangle at (410,475)-(506,501): text "S011: %.0f °C"; shows S011.Deg; alarm colour if S011.Alarm.Adver
rounded rectangle at (510,475)-(561,501): text "MUTE"; alarm colour if TANK.S011_Mute; toggles TANK.S011_Mute
ellipse at (495,245)-(546,271): text "SF009"; alarm colour if SF009.Alarm.Adver
ellipse at (915,170)-(1006,211): text "REDUCED"; invisible if TANK.Reduced = FALSE
rounded rectangle at (550,245)-(601,271): text "BYPASS"; alarm colour if TANK.BypassLevel; toggles TANK.BypassLevel
rounded rectangle at (905,110)-(1016,151): text "CLEAR"; alarm colour if ALARMS.Clear; taps ALARMS.Clear
3 more shapes without text or variables
*)

(* Visualisation VISU_1_WB
rectangle at (785,290)-(891,311): text "LINK UpFwd/DwAft"; invisible if MAIN.fbWB.Manual = FALSE
ellipse at (740,285)-(786,316): invisible if MAIN.fbWB.Manual = FALSE; alarm colour if MAIN.WB_Scoop_Link; toggles MAIN.WB_Scoop_Link
rectangle at (835,205)-(881,226): text "SCOOP"
rectangle at (835,375)-(881,396): text "SCOOP"
polyline at (420,385)-(790,415): alarm colour if MAIN.fbWB_J.SF_Open
polyline at (420,185)-(790,215): alarm colour if MAIN.fbWB_G.SF_Open
polyline at (355,300)-(485,300): alarm colour if MAIN.fbWB.OUT_Pump
ellipse at (390,270)-(451,331): alarm colour if MAIN.fbWB.OUT_Pump
rectangle at (20,550)-(331,601): text "%s"; shows INPUTS.sVisuTime
rounded rectangle at (905,505)-(1016,546): text "RETURN"; opens VISU_0_MAIN
ellipse at (465,95)-(506,136): alarm colour if MAIN.fbWB_A.SF_Open
polyline at (355,135)-(420,150): alarm colour if MAIN.fbWB_D.SF_Open
polyline at (420,135)-(485,150): alarm colour if MAIN.fbWB_A.SF_Open
polyline at (420,220)-(485,300): alarm colour if MAIN.fbWB_F.SF_Open
polyline at (355,220)-(420,300): alarm colour if MAIN.fbWB_E.SF_Open
polyline at (420,185)-(420,220): alarm colour if MAIN.fbWB_E.SF_Open OR MAIN.fbWB_F.SF_Open
polyline at (420,150)-(420,185): alarm colour if MAIN.fbWB_A.SF_Open OR MAIN.fbWB_D.SF_Open
polyline at (240,135)-(240,465): alarm colour if MAIN.fbWB_B.SF_Open OR MAIN.fbWB_I.SF_Open
polyline at (600,135)-(605,465): alarm colour if MAIN.fbWB_C.SF_Open OR MAIN.fbWB_N.SF_Open
polyline at (715,135)-(720,465): alarm colour if MAIN.fbWB_S.SF_Open OR MAIN.fbWB_R.SF_Open
rounded rectangle at (905,110)-(1016,151): text "MANUAL"; alarm colour if MAIN.fbWB.Manual; toggles MAIN.fbWB.Manual
polyline at (420,415)-(420,450): alarm colour if MAIN.fbWB_M.SF_Open OR MAIN.fbWB_K.SF_Open
polyline at (420,380)-(420,415): alarm colour if MAIN.fbWB_H.SF_Open OR MAIN.fbWB_L.SF_Open
polyline at (355,300)-(420,380): alarm colour if MAIN.fbWB_H.SF_Open
polyline at (420,300)-(485,380): alarm colour if MAIN.fbWB_L.SF_Open
polyline at (355,450)-(420,465): alarm colour if MAIN.fbWB_M.SF_Open
polyline at (420,450)-(485,465): alarm colour if MAIN.fbWB_K.SF_Open
ellipse at (335,95)-(376,136): alarm colour if MAIN.fbWB_D.SF_Open
ellipse at (220,95)-(261,136): alarm colour if MAIN.fbWB_B.SF_Open
ellipse at (220,465)-(261,506): alarm colour if MAIN.fbWB_I.SF_Open
ellipse at (490,165)-(531,206): alarm colour if MAIN.fbWB_G.SF_Open
ellipse at (580,95)-(621,136): alarm colour if MAIN.fbWB_C.SF_Open
ellipse at (695,95)-(736,136): alarm colour if MAIN.fbWB_S.SF_Open
polygon at (390,275)-(435,325): text "PUMP"; alarm colour if MAIN.fbWB.OUT_Pump
ellipse at (335,235)-(376,276): alarm colour if MAIN.fbWB_E.SF_Open
ellipse at (465,235)-(506,276): alarm colour if MAIN.fbWB_F.SF_Open
ellipse at (335,325)-(376,366): alarm colour if MAIN.fbWB_H.SF_Open
ellipse at (465,325)-(506,366): alarm colour if MAIN.fbWB_L.SF_Open
ellipse at (490,395)-(531,436): alarm colour if MAIN.fbWB_J.SF_Open
ellipse at (335,465)-(376,506): alarm colour if MAIN.fbWB_M.SF_Open
ellipse at (465,465)-(506,506): alarm colour if MAIN.fbWB_K.SF_Open
ellipse at (580,465)-(621,506): alarm colour if MAIN.fbWB_N.SF_Open
ellipse at (695,465)-(736,506): alarm colour if MAIN.fbWB_R.SF_Open
ellipse at (790,195)-(831,236): alarm colour if MAIN.fbWB_PUD.SF_Open OR MAIN.fbWB_PUD.SF_Half
ellipse at (820,155)-(871,206): invisible if MAIN.fbWB.Manual = FALSE; alarm colour if MAIN.fbWB_PUD.OUT_Open
ellipse at (825,160)-(866,201): text "DW"; invisible if MAIN.fbWB.Manual = FALSE; alarm colour if MAIN.fbWB_PUD.IN_Hmi_Open; taps MAIN.fbWB_PUD.IN_Hmi_Open
ellipse at (750,155)-(801,206): invisible if MAIN.fbWB.Manual = FALSE; alarm colour if MAIN.fbWB_PUD.OUT_Close
ellipse at (755,160)-(796,201): text "UP"; invisible if MAIN.fbWB.Manual = FALSE; alarm colour if MAIN.fbWB_PUD.IN_Hmi_Close; taps MAIN.fbWB_PUD.IN_Hmi_Close
ellipse at (820,225)-(871,276): invisible if MAIN.fbWB.Manual = FALSE; alarm colour if MAIN.fbWB_PAF.OUT_Close
ellipse at (825,230)-(866,271): text "FWD"; invisible if MAIN.fbWB.Manual = FALSE; alarm colour if MAIN.fbWB_PAF.IN_Hmi_Close; taps MAIN.fbWB_PAF.IN_Hmi_Close
ellipse at (750,225)-(801,276): invisible if MAIN.fbWB.Manual = FALSE; alarm colour if MAIN.fbWB_PAF.OUT_Open
ellipse at (755,230)-(796,271): text "AFT"; invisible if MAIN.fbWB.Manual = FALSE; alarm colour if MAIN.fbWB_PAF.IN_Hmi_Open; taps MAIN.fbWB_PAF.IN_Hmi_Open
ellipse at (790,365)-(831,406): alarm colour if MAIN.fbWB_SUD.SF_Open OR MAIN.fbWB_SUD.SF_Half
ellipse at (820,325)-(871,376): invisible if MAIN.fbWB.Manual = FALSE; alarm colour if MAIN.fbWB_SUD.OUT_Open
ellipse at (825,330)-(866,371): text "DW"; invisible if MAIN.fbWB.Manual = FALSE; alarm colour if MAIN.fbWB_SUD.IN_Hmi_Open; taps MAIN.fbWB_SUD.IN_Hmi_Open
ellipse at (750,325)-(801,376): invisible if MAIN.fbWB.Manual = FALSE; alarm colour if MAIN.fbWB_SUD.OUT_Close
ellipse at (755,330)-(796,371): text "UP"; invisible if MAIN.fbWB.Manual = FALSE; alarm colour if MAIN.fbWB_SUD.IN_Hmi_Close; taps MAIN.fbWB_SUD.IN_Hmi_Close
ellipse at (820,395)-(871,446): invisible if MAIN.fbWB.Manual = FALSE; alarm colour if MAIN.fbWB_SAF.OUT_Close
ellipse at (825,400)-(866,441): text "FWD"; invisible if MAIN.fbWB.Manual = FALSE; alarm colour if MAIN.fbWB_SAF.IN_Hmi_Close; taps MAIN.fbWB_SAF.IN_Hmi_Close
ellipse at (750,395)-(801,446): invisible if MAIN.fbWB.Manual = FALSE; alarm colour if MAIN.fbWB_SAF.OUT_Open
rounded rectangle at (900,50)-(1021,101): alarm colour if MAIN.aHP_Enable[19]
rounded rectangle at (905,55)-(1016,96): text "ENABLE"; alarm colour if MAIN.aHP_Enable[19]; toggles MAIN.aHP_Enable[19]
rectangle at (40,510)-(121,531): text "%.0f bar"; shows P2500.Bar; alarm colour if P2500.Alarm.Adver; runs INTERN ASSIGN INPUTS.PresSelCalStbd[9]:=(FALSE)
rectangle at (40,495)-(111,511): text "P2500"
ellipse at (230,100)-(251,131): text "B"; alarm colour if MAIN.fbWB_B.SF_Close
ellipse at (185,90)-(236,141): invisible if MAIN.fbWB.Manual = FALSE; alarm colour if MAIN.fbWB_B.OUT_Close
ellipse at (190,95)-(231,136): text "CLOSE"; invisible if MAIN.fbWB.Manual = FALSE; alarm colour if MAIN.fbWB_B.IN_Hmi_Close; taps MAIN.fbWB_B.IN_Hmi_Close
ellipse at (345,100)-(366,131): text "D"; alarm colour if MAIN.fbWB_D.SF_Close
ellipse at (475,100)-(496,131): text "A"; alarm colour if MAIN.fbWB_A.SF_Close
ellipse at (590,100)-(611,131): text "C"; alarm colour if MAIN.fbWB_C.SF_Close
ellipse at (705,100)-(726,131): text "S"; alarm colour if MAIN.fbWB_S.SF_Close
ellipse at (345,240)-(366,271): text "E"; alarm colour if MAIN.fbWB_E.SF_Close
ellipse at (500,170)-(521,201): text "G"; alarm colour if MAIN.fbWB_G.SF_Close
ellipse at (475,240)-(496,271): text "F"; alarm colour if MAIN.fbWB_F.SF_Close
ellipse at (345,330)-(366,361): text "H"; alarm colour if MAIN.fbWB_H.SF_Close
ellipse at (475,330)-(496,361): text "L"; alarm colour if MAIN.fbWB_L.SF_Close
ellipse at (500,400)-(521,431): text "J"; alarm colour if MAIN.fbWB_J.SF_Close
ellipse at (230,470)-(251,501): text "I"; alarm colour if MAIN.fbWB_I.SF_Close
ellipse at (345,470)-(366,501): text "M"; alarm colour if MAIN.fbWB_M.SF_Close
ellipse at (475,470)-(496,501): text "K"; alarm colour if MAIN.fbWB_K.SF_Close
ellipse at (590,470)-(611,501): text "N"; alarm colour if MAIN.fbWB_N.SF_Close
ellipse at (705,470)-(726,501): text "R"; alarm colour if MAIN.fbWB_R.SF_Close
ellipse at (185,460)-(236,511): invisible if MAIN.fbWB.Manual = FALSE; alarm colour if MAIN.fbWB_I.OUT_Close
ellipse at (190,465)-(231,506): text "CLOSE"; invisible if MAIN.fbWB.Manual = FALSE; alarm colour if MAIN.fbWB_I.IN_Hmi_Close; taps MAIN.fbWB_I.IN_Hmi_Close
ellipse at (300,90)-(351,141): invisible if MAIN.fbWB.Manual = FALSE; alarm colour if MAIN.fbWB_D.OUT_Close
ellipse at (305,95)-(346,136): text "CLOSE"; invisible if MAIN.fbWB.Manual = FALSE; alarm colour if MAIN.fbWB_D.IN_Hmi_Close; taps MAIN.fbWB_D.IN_Hmi_Close
ellipse at (245,90)-(296,141): invisible if MAIN.fbWB.Manual = FALSE; alarm colour if MAIN.fbWB_B.OUT_Open
ellipse at (250,95)-(291,136): text "OPEN"; invisible if MAIN.fbWB.Manual = FALSE; alarm colour if MAIN.fbWB_B.IN_Hmi_Open; taps MAIN.fbWB_B.IN_Hmi_Open
ellipse at (300,460)-(351,511): invisible if MAIN.fbWB.Manual = FALSE; alarm colour if MAIN.fbWB_M.OUT_Close
ellipse at (305,465)-(346,506): text "CLOSE"; invisible if MAIN.fbWB.Manual = FALSE; alarm colour if MAIN.fbWB_M.IN_Hmi_Close; taps MAIN.fbWB_M.IN_Hmi_Close
ellipse at (245,460)-(296,511): invisible if MAIN.fbWB.Manual = FALSE; alarm colour if MAIN.fbWB_I.OUT_Open
ellipse at (250,465)-(291,506): text "OPEN"; invisible if MAIN.fbWB.Manual = FALSE; alarm colour if MAIN.fbWB_I.IN_Hmi_Open; taps MAIN.fbWB_I.IN_Hmi_Open
ellipse at (430,460)-(481,511): invisible if MAIN.fbWB.Manual = FALSE; alarm colour if MAIN.fbWB_K.OUT_Close
ellipse at (435,465)-(476,506): text "CLOSE"; invisible if MAIN.fbWB.Manual = FALSE; alarm colour if MAIN.fbWB_K.IN_Hmi_Close; taps MAIN.fbWB_K.IN_Hmi_Close
ellipse at (360,460)-(411,511): invisible if MAIN.fbWB.Manual = FALSE; alarm colour if MAIN.fbWB_M.OUT_Open
ellipse at (365,465)-(406,506): text "OPEN"; invisible if MAIN.fbWB.Manual = FALSE; alarm colour if MAIN.fbWB_M.IN_Hmi_Open; taps MAIN.fbWB_M.IN_Hmi_Open
ellipse at (545,460)-(596,511): invisible if MAIN.fbWB.Manual = FALSE; alarm colour if MAIN.fbWB_N.OUT_Close
ellipse at (550,465)-(591,506): text "CLOSE"; invisible if MAIN.fbWB.Manual = FALSE; alarm colour if MAIN.fbWB_N.IN_Hmi_Close; taps MAIN.fbWB_N.IN_Hmi_Close
ellipse at (490,460)-(541,511): invisible if MAIN.fbWB.Manual = FALSE; alarm colour if MAIN.fbWB_K.OUT_Open
ellipse at (495,465)-(536,506): text "OPEN"; invisible if MAIN.fbWB.Manual = FALSE; alarm colour if MAIN.fbWB_K.IN_Hmi_Open; taps MAIN.fbWB_K.IN_Hmi_Open
ellipse at (720,460)-(771,511): invisible if MAIN.fbWB.Manual = FALSE; alarm colour if MAIN.fbWB_R.OUT_Open
ellipse at (725,465)-(766,506): text "OPEN"; invisible if MAIN.fbWB.Manual = FALSE; alarm colour if MAIN.fbWB_R.IN_Hmi_Open; taps MAIN.fbWB_R.IN_Hmi_Open
ellipse at (755,400)-(796,441): text "AFT"; invisible if MAIN.fbWB.Manual = FALSE; alarm colour if MAIN.fbWB_SAF.IN_Hmi_Open; taps MAIN.fbWB_SAF.IN_Hmi_Open
ellipse at (660,460)-(711,511): invisible if MAIN.fbWB.Manual = FALSE; alarm colour if MAIN.fbWB_R.OUT_Close
ellipse at (665,465)-(706,506): text "CLOSE"; invisible if MAIN.fbWB.Manual = FALSE; alarm colour if MAIN.fbWB_R.IN_Hmi_Close; taps MAIN.fbWB_R.IN_Hmi_Close
ellipse at (605,460)-(656,511): invisible if MAIN.fbWB.Manual = FALSE; alarm colour if MAIN.fbWB_N.OUT_Open
ellipse at (610,465)-(651,506): text "OPEN"; invisible if MAIN.fbWB.Manual = FALSE; alarm colour if MAIN.fbWB_N.IN_Hmi_Open; taps MAIN.fbWB_N.IN_Hmi_Open
ellipse at (515,160)-(566,211): invisible if MAIN.fbWB.Manual = FALSE; alarm colour if MAIN.fbWB_G.OUT_Open
ellipse at (520,165)-(561,206): text "OPEN"; invisible if MAIN.fbWB.Manual = FALSE; alarm colour if MAIN.fbWB_G.IN_Hmi_Open; taps MAIN.fbWB_G.IN_Hmi_Open
ellipse at (515,390)-(566,441): invisible if MAIN.fbWB.Manual = FALSE; alarm colour if MAIN.fbWB_J.OUT_Open
ellipse at (520,395)-(561,436): text "OPEN"; invisible if MAIN.fbWB.Manual = FALSE; alarm colour if MAIN.fbWB_J.IN_Hmi_Open; taps MAIN.fbWB_J.IN_Hmi_Open
ellipse at (455,160)-(506,211): invisible if MAIN.fbWB.Manual = FALSE; alarm colour if MAIN.fbWB_G.OUT_Close
ellipse at (460,165)-(501,206): text "CLOSE"; invisible if MAIN.fbWB.Manual = FALSE; alarm colour if MAIN.fbWB_G.IN_Hmi_Close; taps MAIN.fbWB_G.IN_Hmi_Close
ellipse at (455,390)-(506,441): invisible if MAIN.fbWB.Manual = FALSE; alarm colour if MAIN.fbWB_J.OUT_Close
ellipse at (460,395)-(501,436): text "CLOSE"; invisible if MAIN.fbWB.Manual = FALSE; alarm colour if MAIN.fbWB_J.IN_Hmi_Close; taps MAIN.fbWB_J.IN_Hmi_Close
ellipse at (490,230)-(541,281): invisible if MAIN.fbWB.Manual = FALSE; alarm colour if MAIN.fbWB_F.OUT_Open
ellipse at (495,235)-(536,276): text "OPEN"; invisible if MAIN.fbWB.Manual = FALSE; alarm colour if MAIN.fbWB_F.IN_Hmi_Open; taps MAIN.fbWB_F.IN_Hmi_Open
ellipse at (490,320)-(541,371): invisible if MAIN.fbWB.Manual = FALSE; alarm colour if MAIN.fbWB_L.OUT_Open
ellipse at (495,325)-(536,366): text "OPEN"; invisible if MAIN.fbWB.Manual = FALSE; alarm colour if MAIN.fbWB_L.IN_Hmi_Open; taps MAIN.fbWB_L.IN_Hmi_Open
ellipse at (430,230)-(481,281): invisible if MAIN.fbWB.Manual = FALSE; alarm colour if MAIN.fbWB_F.OUT_Close
ellipse at (435,235)-(476,276): text "CLOSE"; invisible if MAIN.fbWB.Manual = FALSE; alarm colour if MAIN.fbWB_F.IN_Hmi_Close; taps MAIN.fbWB_F.IN_Hmi_Close
ellipse at (430,320)-(481,371): invisible if MAIN.fbWB.Manual = FALSE; alarm colour if MAIN.fbWB_L.OUT_Close
ellipse at (435,325)-(476,366): text "CLOSE"; invisible if MAIN.fbWB.Manual = FALSE; alarm colour if MAIN.fbWB_L.IN_Hmi_Close; taps MAIN.fbWB_L.IN_Hmi_Close
ellipse at (360,230)-(411,281): invisible if MAIN.fbWB.Manual = FALSE; alarm colour if MAIN.fbWB_E.OUT_Open
ellipse at (365,235)-(406,276): text "OPEN"; invisible if MAIN.fbWB.Manual = FALSE; alarm colour if MAIN.fbWB_E.IN_Hmi_Open; taps MAIN.fbWB_E.IN_Hmi_Open
ellipse at (360,320)-(411,371): invisible if MAIN.fbWB.Manual = FALSE; alarm colour if MAIN.fbWB_H.OUT_Open
ellipse at (365,325)-(406,366): text "OPEN"; invisible if MAIN.fbWB.Manual = FALSE; alarm colour if MAIN.fbWB_H.IN_Hmi_Open; taps MAIN.fbWB_H.IN_Hmi_Open
ellipse at (300,230)-(351,281): invisible if MAIN.fbWB.Manual = FALSE; alarm colour if MAIN.fbWB_E.OUT_Close
ellipse at (305,235)-(346,276): text "CLOSE"; invisible if MAIN.fbWB.Manual = FALSE; alarm colour if MAIN.fbWB_E.IN_Hmi_Close; taps MAIN.fbWB_E.IN_Hmi_Close
ellipse at (300,320)-(351,371): invisible if MAIN.fbWB.Manual = FALSE; alarm colour if MAIN.fbWB_H.OUT_Close
ellipse at (305,325)-(346,366): text "CLOSE"; invisible if MAIN.fbWB.Manual = FALSE; alarm colour if MAIN.fbWB_H.IN_Hmi_Close; taps MAIN.fbWB_H.IN_Hmi_Close
ellipse at (430,90)-(481,141): invisible if MAIN.fbWB.Manual = FALSE; alarm colour if MAIN.fbWB_A.OUT_Close
ellipse at (435,95)-(476,136): text "CLOSE"; invisible if MAIN.fbWB.Manual = FALSE; alarm colour if MAIN.fbWB_A.IN_Hmi_Close; taps MAIN.fbWB_A.IN_Hmi_Close
ellipse at (360,90)-(411,141): invisible if MAIN.fbWB.Manual = FALSE; alarm colour if MAIN.fbWB_D.OUT_Open
ellipse at (365,95)-(406,136): text "OPEN"; invisible if MAIN.fbWB.Manual = FALSE; alarm colour if MAIN.fbWB_D.IN_Hmi_Open; taps MAIN.fbWB_D.IN_Hmi_Open
ellipse at (545,90)-(596,141): invisible if MAIN.fbWB.Manual = FALSE; alarm colour if MAIN.fbWB_C.OUT_Close
ellipse at (550,95)-(591,136): text "CLOSE"; invisible if MAIN.fbWB.Manual = FALSE; alarm colour if MAIN.fbWB_C.IN_Hmi_Close; taps MAIN.fbWB_C.IN_Hmi_Close
ellipse at (490,90)-(541,141): invisible if MAIN.fbWB.Manual = FALSE; alarm colour if MAIN.fbWB_A.OUT_Open
ellipse at (495,95)-(536,136): text "OPEN"; invisible if MAIN.fbWB.Manual = FALSE; alarm colour if MAIN.fbWB_A.IN_Hmi_Open; taps MAIN.fbWB_A.IN_Hmi_Open
ellipse at (660,90)-(711,141): invisible if MAIN.fbWB.Manual = FALSE; alarm colour if MAIN.fbWB_S.OUT_Close
ellipse at (665,95)-(706,136): text "CLOSE"; invisible if MAIN.fbWB.Manual = FALSE; alarm colour if MAIN.fbWB_S.IN_Hmi_Close; taps MAIN.fbWB_S.IN_Hmi_Close
ellipse at (605,90)-(656,141): invisible if MAIN.fbWB.Manual = FALSE; alarm colour if MAIN.fbWB_C.OUT_Open
ellipse at (610,95)-(651,136): text "OPEN"; invisible if MAIN.fbWB.Manual = FALSE; alarm colour if MAIN.fbWB_C.IN_Hmi_Open; taps MAIN.fbWB_C.IN_Hmi_Open
ellipse at (720,90)-(771,141): invisible if MAIN.fbWB.Manual = FALSE; alarm colour if MAIN.fbWB_S.OUT_Open
ellipse at (725,95)-(766,136): text "OPEN"; invisible if MAIN.fbWB.Manual = FALSE; alarm colour if MAIN.fbWB_S.IN_Hmi_Open; taps MAIN.fbWB_S.IN_Hmi_Open
rounded rectangle at (905,450)-(1016,491): text "CONFIG: / WB"; opens VISU_CFG_WB
rounded rectangle at (905,395)-(1016,436): text "CALIB: / WB"; opens VISU_CAL_WB
rectangle at (20,0)-(331,51): text "WATER BALLAST"
rounded rectangle at (260,55)-(331,71): text "AFT PORT"; alarm colour if SF021
rounded rectangle at (565,55)-(636,71): text "FWR PORT"; alarm colour if SF022
ellipse at (620,265)-(691,336): invisible if MAIN.fbWB.Manual = FALSE; alarm colour if MAIN.fbWB.OUT_Pump
ellipse at (630,275)-(681,326): text "PUMP"; invisible if MAIN.fbWB.Manual = FALSE; alarm colour if MAIN.fbWB.IN_Hmi_Pump; taps MAIN.fbWB.IN_Hmi_Pump
rounded rectangle at (565,530)-(636,546): text "FWR STBD"; alarm colour if SF024
rounded rectangle at (260,530)-(331,546): text "AFT STBD"; alarm colour if SF023
ellipse at (800,200)-(821,231): text "SC"; alarm colour if MAIN.fbWB_PUD.SF_Close
polygon at (800,240)-(810,260): alarm colour if MAIN.fbWB_PAF.SF_Open
polygon at (810,240)-(820,260): alarm colour if MAIN.fbWB_PAF.SF_Close
polygon at (800,410)-(810,430): alarm colour if MAIN.fbWB_SAF.SF_Open
polygon at (810,410)-(820,430): alarm colour if MAIN.fbWB_SAF.SF_Close
ellipse at (800,175)-(821,196): text "1/2"; alarm colour if MAIN.fbWB_PUD.SF_Half
ellipse at (800,345)-(821,366): text "1/2"; alarm colour if MAIN.fbWB_SUD.SF_Half
ellipse at (800,370)-(821,401): text "SC"; alarm colour if MAIN.fbWB_SUD.SF_Close
ellipse at (15,70)-(86,141): alarm colour if MAIN.fbWB.OUT_P_Fwd
ellipse at (25,80)-(76,131): text "FWD"; alarm colour if MAIN.fbWB.IN_Hmi_P_Fwd; taps MAIN.fbWB.IN_Hmi_P_Fwd
ellipse at (95,70)-(166,141): alarm colour if MAIN.fbWB.OUT_P_Aft
ellipse at (105,80)-(156,131): text "AFT"; alarm colour if MAIN.fbWB.IN_Hmi_P_Aft; taps MAIN.fbWB.IN_Hmi_P_Aft
ellipse at (15,150)-(86,221): alarm colour if MAIN.fbWB.OUT_S_Fwd
ellipse at (25,160)-(76,211): text "FWD"; alarm colour if MAIN.fbWB.IN_Hmi_S_Fwd; taps MAIN.fbWB.IN_Hmi_S_Fwd
ellipse at (95,150)-(166,221): alarm colour if MAIN.fbWB.OUT_S_Aft
ellipse at (105,160)-(156,211): text "AFT"; alarm colour if MAIN.fbWB.IN_Hmi_S_Aft; taps MAIN.fbWB.IN_Hmi_S_Aft
rounded rectangle at (630,340)-(681,371): text "%d %%"; shows MAIN.fbWB.IN_Hmi_Pump_Perc; invisible if MAIN.fbWB.Manual = FALSE; editable 5..100
ellipse at (15,245)-(86,316): alarm colour if MAIN.fbWB.OUT_Fill
ellipse at (25,255)-(76,306): text "FILL"; alarm colour if MAIN.fbWB.IN_Hmi_Fill; taps MAIN.fbWB.IN_Hmi_Fill
ellipse at (95,245)-(166,316): alarm colour if MAIN.fbWB.OUT_12
ellipse at (105,255)-(156,306): text "1/2 / SCOOP"; alarm colour if MAIN.fbWB.IN_Hmi_12; taps MAIN.fbWB.IN_Hmi_12
ellipse at (15,405)-(86,476): alarm colour if MAIN.fbWB.OUT_Dump
ellipse at (25,415)-(76,466): text "DUMP"; alarm colour if MAIN.fbWB.IN_Hmi_Dump; taps MAIN.fbWB.IN_Hmi_Dump
ellipse at (95,405)-(166,476): alarm colour if MAIN.fbWB.OUT_Move
ellipse at (105,415)-(156,466): text "MOVE"; alarm colour if MAIN.fbWB.IN_Hmi_Move; taps MAIN.fbWB.IN_Hmi_Move
ellipse at (55,325)-(126,396): alarm colour if MAIN.fbWB.OUT_Stop
ellipse at (65,335)-(116,386): text "STOP"; alarm colour if MAIN.fbWB.IN_Hmi_Stop; taps MAIN.fbWB.IN_Hmi_Stop
rectangle at (0,0)-(1,1): text "{ExtendedElement},Visu\ElementDLL.ete,1,@Bargraph,246,21,3,0,1,LS021.Pos,,%,25,50,0,100,0,0,0,0,0,0,0,-13,16,700,Arial,0,255,0,255,0,0,0,0,0,0,0,0,0,,0,"
rectangle at (123,0)-(247,21): alarm colour if (LS021.Pos) < 0; left ((LS021.Pos * 1.0) - 50)  * -2.46
rectangle at (0,0)-(1,1): text "{ExtendedElement},Visu\ElementDLL.ete,1,@Bargraph,246,21,3,0,1,LS023.Pos,,%,25,50,0,100,0,0,0,0,0,0,0,-13,16,700,Arial,0,255,0,255,0,0,0,0,0,0,0,0,0,,0,"
rectangle at (123,0)-(247,21): alarm colour if (LS023.Pos) < 0; left ((LS023.Pos * 1.0) - 50)  * -2.46
rectangle at (490,290)-(591,311): text "EVP1609: %d %%"; shows EVP1608_9 / 10; alarm colour if EVP1608_9 = 0
rectangle at (0,0)-(1,1): text "{ExtendedElement},Visu\ElementDLL.ete,1,@Bargraph,371,21,3,0,1,LS022.Pos,,%,25,50,0,100,0,0,0,0,0,0,0,-13,16,700,Arial,0,255,0,255,0,0,0,0,0,0,0,0,0,,0,"
rectangle at (186,0)-(372,21): alarm colour if (LS022.Pos) < 0; left ((LS022.Pos * 1.0) - 50)  * -3.7
rectangle at (0,0)-(1,1): text "{ExtendedElement},Visu\ElementDLL.ete,1,@Bargraph,371,21,3,0,1,LS024.Pos,,%,25,50,0,100,0,0,0,0,0,0,0,-13,16,700,Arial,0,255,0,255,0,0,0,0,0,0,0,0,0,,0,"
rectangle at (186,0)-(372,21): alarm colour if (LS024.Pos) < 0; left ((LS024.Pos * 1.0) - 50)  * -3.7
ellipse at (800,155)-(821,176): text "100"; alarm colour if MAIN.fbWB_PUD.SF_Open
ellipse at (800,325)-(821,346): text "100"; alarm colour if MAIN.fbWB_SUD.SF_Open
other_PIE at (755,300)-(755,300): invisible if MAIN.fbWB.Manual = FALSE
other_PIE at (770,300)-(770,300): invisible if MAIN.fbWB.Manual = FALSE
ellipse at (905,165)-(1016,206): text "ERROR: / %d"; shows MAIN.fbWB.Error; invisible if MAIN.fbWB.Error = 0
10 more shapes without text or variables
*)

(* Visualisation VISU_1_WINCHES
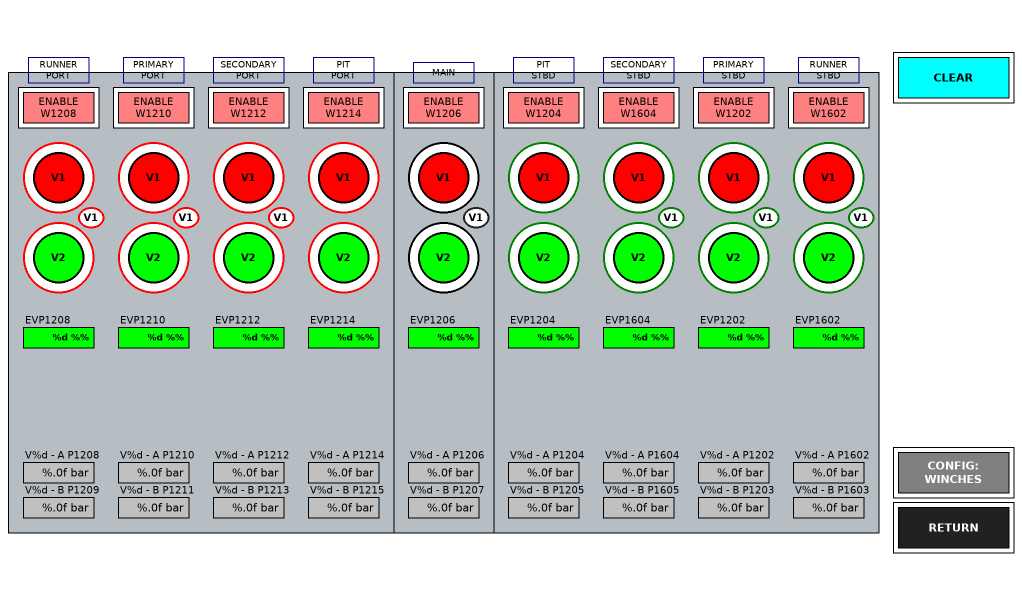
rectangle at (20,550)-(331,601): text "%s"; shows INPUTS.sVisuTime
rounded rectangle at (905,505)-(1016,546): text "RETURN"; opens VISU_0_MAIN
rectangle at (20,0)-(331,51): text "WINCHES"
ellipse at (705,140)-(776,211): alarm colour if MAIN.fbW1202.OUT_1
ellipse at (705,220)-(776,291): alarm colour if MAIN.fbW1202.OUT_2
ellipse at (715,150)-(766,201): text "V1"; alarm colour if MAIN.fbW1202.IN_Hmi_1; taps MAIN.fbW1202.IN_Hmi_1
ellipse at (715,230)-(766,281): text "V2"; alarm colour if MAIN.fbW1202.IN_Hmi_2; taps MAIN.fbW1202.IN_Hmi_2
rounded rectangle at (905,450)-(1016,491): text "CONFIG: / WINCHES"; opens VISU_CFG_WINCHES
ellipse at (515,140)-(586,211): alarm colour if MAIN.fbW1204.OUT_1
ellipse at (515,220)-(586,291): alarm colour if MAIN.fbW1204.OUT_2
ellipse at (525,150)-(576,201): text "V1"; alarm colour if MAIN.fbW1204.IN_Hmi_1; taps MAIN.fbW1204.IN_Hmi_1
ellipse at (525,230)-(576,281): text "V2"; alarm colour if MAIN.fbW1204.IN_Hmi_2; taps MAIN.fbW1204.IN_Hmi_2
rectangle at (515,460)-(586,481): text "%.0f bar"; shows P1204.Bar; alarm colour if P1204.Alarm.Adver; runs INTERN ASSIGN INPUTS.PresSelCalStbd[9]:=(FALSE)
rectangle at (515,445)-(586,461): text "V%d - A P1204"; shows MAIN.fbW1204.SpdA
rectangle at (515,480)-(586,496): text "V%d - B P1205"; shows MAIN.fbW1204.SpdB
rectangle at (515,495)-(586,516): text "%.0f bar"; shows P1205.Bar; alarm colour if P1205.Alarm.Adver; runs INTERN ASSIGN INPUTS.PresSelCalStbd[9]:=(FALSE)
rectangle at (705,460)-(776,481): text "%.0f bar"; shows P1202.Bar; alarm colour if P1202.Alarm.Adver; runs INTERN ASSIGN INPUTS.PresSelCalStbd[9]:=(FALSE)
rectangle at (705,445)-(776,461): text "V%d - A P1202"; shows MAIN.fbW1202.SpdA
rectangle at (705,480)-(776,496): text "V%d - B P1203"; shows MAIN.fbW1202.SpdB
rectangle at (705,495)-(776,516): text "%.0f bar"; shows P1203.Bar; alarm colour if P1203.Alarm.Adver; runs INTERN ASSIGN INPUTS.PresSelCalStbd[9]:=(FALSE)
rounded rectangle at (705,90)-(776,121): text "ENABLE / W1202"; alarm colour if MAIN.aLP_Enable[4]; toggles MAIN.aLP_Enable[4]
rounded rectangle at (515,90)-(586,121): text "ENABLE / W1204"; alarm colour if MAIN.aLP_Enable[5]; toggles MAIN.aLP_Enable[5]
rounded rectangle at (415,90)-(486,121): text "ENABLE / W1206"; alarm colour if MAIN.aLP_Enable[6]; toggles MAIN.aLP_Enable[6]
rounded rectangle at (30,90)-(101,121): text "ENABLE / W1208"; alarm colour if MAIN.aLP_Enable[7]; toggles MAIN.aLP_Enable[7]
rounded rectangle at (125,90)-(196,121): text "ENABLE / W1210"; alarm colour if MAIN.aLP_Enable[8]; toggles MAIN.aLP_Enable[8]
rounded rectangle at (220,90)-(291,121): text "ENABLE / W1212"; alarm colour if MAIN.aLP_Enable[9]; toggles MAIN.aLP_Enable[9]
rounded rectangle at (315,90)-(386,121): text "ENABLE / W1214"; alarm colour if MAIN.aLP_Enable[10]; toggles MAIN.aLP_Enable[10]
rounded rectangle at (800,90)-(871,121): text "ENABLE / W1602"; alarm colour if MAIN.aLP_Enable[14]; toggles MAIN.aLP_Enable[14]
rounded rectangle at (610,90)-(681,121): text "ENABLE / W1604"; alarm colour if MAIN.aLP_Enable[15]; toggles MAIN.aLP_Enable[15]
rectangle at (520,55)-(581,81): text "PIT / STBD"
rectangle at (705,325)-(776,346): text "%d %%"; shows EVP1202_3 / 10; alarm colour if EVP1202_3 = 0
rectangle at (515,325)-(586,346): text "%d %%"; shows EVP1204_5 / 10; alarm colour if EVP1204_5 = 0
rectangle at (705,310)-(776,326): text "EVP1202"
rectangle at (515,310)-(586,326): text "EVP1204"
ellipse at (415,140)-(486,211): alarm colour if MAIN.fbW1206.OUT_1
ellipse at (415,220)-(486,291): alarm colour if MAIN.fbW1206.OUT_2
ellipse at (425,150)-(476,201): text "V1"; alarm colour if MAIN.fbW1206.IN_Hmi_1; taps MAIN.fbW1206.IN_Hmi_1
ellipse at (425,230)-(476,281): text "V2"; alarm colour if MAIN.fbW1206.IN_Hmi_2; taps MAIN.fbW1206.IN_Hmi_2
ellipse at (30,140)-(101,211): alarm colour if MAIN.fbW1208.OUT_1
ellipse at (30,220)-(101,291): alarm colour if MAIN.fbW1208.OUT_2
ellipse at (40,150)-(91,201): text "V1"; alarm colour if MAIN.fbW1208.IN_Hmi_1; taps MAIN.fbW1208.IN_Hmi_1
ellipse at (40,230)-(91,281): text "V2"; alarm colour if MAIN.fbW1208.IN_Hmi_2; taps MAIN.fbW1208.IN_Hmi_2
rectangle at (420,60)-(481,81): text "MAIN"
rectangle at (30,460)-(101,481): text "%.0f bar"; shows P1208.Bar; alarm colour if P1208.Alarm.Adver; runs INTERN ASSIGN INPUTS.PresSelCalStbd[9]:=(FALSE)
rectangle at (30,445)-(106,461): text "V%d - A P1208"; shows MAIN.fbW1208.SpdA
rectangle at (30,480)-(106,496): text "V%d - B P1209"; shows MAIN.fbW1208.SpdB
rectangle at (30,495)-(101,516): text "%.0f bar"; shows P1209.Bar; alarm colour if P1209.Alarm.Adver; runs INTERN ASSIGN INPUTS.PresSelCalStbd[9]:=(FALSE)
rectangle at (415,460)-(486,481): text "%.0f bar"; shows P1206.Bar; alarm colour if P1206.Alarm.Adver; runs INTERN ASSIGN INPUTS.PresSelCalStbd[9]:=(FALSE)
rectangle at (415,445)-(486,461): text "V%d - A P1206"; shows MAIN.fbW1206.SpdA
rectangle at (415,480)-(486,496): text "V%d - B P1207"; shows MAIN.fbW1206.SpdB
rectangle at (415,495)-(486,516): text "%.0f bar"; shows P1207.Bar; alarm colour if P1207.Alarm.Adver; runs INTERN ASSIGN INPUTS.PresSelCalStbd[9]:=(FALSE)
rectangle at (35,55)-(96,81): text "RUNNER / PORT"
rectangle at (415,325)-(486,346): text "%d %%"; shows EVP1206_7 / 10; alarm colour if EVP1206_7 = 0
rectangle at (30,325)-(101,346): text "%d %%"; shows EVP1208_9 / 10; alarm colour if EVP1208_9 = 0
rectangle at (415,310)-(486,326): text "EVP1206"
rectangle at (30,310)-(101,326): text "EVP1208"
ellipse at (220,140)-(291,211): alarm colour if MAIN.fbW1212.OUT_1
ellipse at (220,220)-(291,291): alarm colour if MAIN.fbW1212.OUT_2
ellipse at (230,150)-(281,201): text "V1"; alarm colour if MAIN.fbW1212.IN_Hmi_1; taps MAIN.fbW1212.IN_Hmi_1
ellipse at (230,230)-(281,281): text "V2"; alarm colour if MAIN.fbW1212.IN_Hmi_2; taps MAIN.fbW1212.IN_Hmi_2
ellipse at (315,140)-(386,211): alarm colour if MAIN.fbW1214.OUT_1
ellipse at (315,220)-(386,291): alarm colour if MAIN.fbW1214.OUT_2
ellipse at (325,150)-(376,201): text "V1"; alarm colour if MAIN.fbW1214.IN_Hmi_1; taps MAIN.fbW1214.IN_Hmi_1
ellipse at (325,230)-(376,281): text "V2"; alarm colour if MAIN.fbW1214.IN_Hmi_2; taps MAIN.fbW1214.IN_Hmi_2
rectangle at (315,460)-(386,481): text "%.0f bar"; shows P1214.Bar; alarm colour if P1214.Alarm.Adver; runs INTERN ASSIGN INPUTS.PresSelCalStbd[9]:=(FALSE)
rectangle at (315,445)-(386,461): text "V%d - A P1214"; shows MAIN.fbW1214.SpdA
rectangle at (315,480)-(386,496): text "V%d - B P1215"; shows MAIN.fbW1214.SpdB
rectangle at (315,495)-(386,516): text "%.0f bar"; shows P1215.Bar; alarm colour if P1215.Alarm.Adver; runs INTERN ASSIGN INPUTS.PresSelCalStbd[9]:=(FALSE)
rectangle at (220,460)-(291,481): text "%.0f bar"; shows P1212.Bar; alarm colour if P1212.Alarm.Adver; runs INTERN ASSIGN INPUTS.PresSelCalStbd[9]:=(FALSE)
rectangle at (220,445)-(291,461): text "V%d - A P1212"; shows MAIN.fbW1212.SpdA
rectangle at (220,480)-(291,496): text "V%d - B P1213"; shows MAIN.fbW1212.SpdB
rectangle at (220,495)-(291,516): text "%.0f bar"; shows P1213.Bar; alarm colour if P1213.Alarm.Adver; runs INTERN ASSIGN INPUTS.PresSelCalStbd[9]:=(FALSE)
rectangle at (320,55)-(381,81): text "PIT / PORT"
rectangle at (220,325)-(291,346): text "%d %%"; shows EVP1212_3 / 10; alarm colour if EVP1212_3 = 0
rectangle at (315,325)-(386,346): text "%d %%"; shows EVP1214_5 / 10; alarm colour if EVP1214_5 = 0
rectangle at (220,310)-(291,326): text "EVP1212"
rectangle at (315,310)-(386,326): text "EVP1214"
ellipse at (800,140)-(871,211): alarm colour if MAIN.fbW1602.OUT_1
ellipse at (800,220)-(871,291): alarm colour if MAIN.fbW1602.OUT_2
ellipse at (810,150)-(861,201): text "V1"; alarm colour if MAIN.fbW1602.IN_Hmi_1; taps MAIN.fbW1602.IN_Hmi_1
ellipse at (810,230)-(861,281): text "V2"; alarm colour if MAIN.fbW1602.IN_Hmi_2; taps MAIN.fbW1602.IN_Hmi_2
ellipse at (610,140)-(681,211): alarm colour if MAIN.fbW1604.OUT_1
ellipse at (610,220)-(681,291): alarm colour if MAIN.fbW1604.OUT_2
ellipse at (620,150)-(671,201): text "V1"; alarm colour if MAIN.fbW1604.IN_Hmi_1; taps MAIN.fbW1604.IN_Hmi_1
ellipse at (620,230)-(671,281): text "V2"; alarm colour if MAIN.fbW1604.IN_Hmi_2; taps MAIN.fbW1604.IN_Hmi_2
rectangle at (805,55)-(866,81): text "RUNNER / STBD"
rectangle at (610,460)-(681,481): text "%.0f bar"; shows P1604.Bar; alarm colour if P1604.Alarm.Adver; runs INTERN ASSIGN INPUTS.PresSelCalStbd[9]:=(FALSE)
rectangle at (610,445)-(681,461): text "V%d - A P1604"; shows MAIN.fbW1604.SpdA
rectangle at (610,480)-(681,496): text "V%d - B P1605"; shows MAIN.fbW1604.SpdB
rectangle at (610,495)-(681,516): text "%.0f bar"; shows P1605.Bar; alarm colour if P1605.Alarm.Adver; runs INTERN ASSIGN INPUTS.PresSelCalStbd[9]:=(FALSE)
rectangle at (800,460)-(871,481): text "%.0f bar"; shows P1602.Bar; alarm colour if P1602.Alarm.Adver; runs INTERN ASSIGN INPUTS.PresSelCalStbd[9]:=(FALSE)
rectangle at (800,445)-(871,461): text "V%d - A P1602"; shows MAIN.fbW1602.SpdA
rectangle at (800,480)-(881,496): text "V%d - B P1603"; shows MAIN.fbW1602.SpdB
rectangle at (800,495)-(871,516): text "%.0f bar"; shows P1603.Bar; alarm colour if P1603.Alarm.Adver; runs INTERN ASSIGN INPUTS.PresSelCalStbd[9]:=(FALSE)
rectangle at (610,55)-(681,81): text "SECONDARY / STBD"
rectangle at (800,325)-(871,346): text "%d %%"; shows EVP1602_3 / 10; alarm colour if EVP1602_3 = 0
rectangle at (610,325)-(681,346): text "%d %%"; shows EVP1604_5 / 10; alarm colour if EVP1604_5 = 0
rectangle at (800,310)-(871,326): text "EVP1602"
rectangle at (610,310)-(681,326): text "EVP1604"
ellipse at (125,140)-(196,211): alarm colour if MAIN.fbW1210.OUT_1
ellipse at (125,220)-(196,291): alarm colour if MAIN.fbW1210.OUT_2
ellipse at (135,150)-(186,201): text "V1"; alarm colour if MAIN.fbW1210.IN_Hmi_1; taps MAIN.fbW1210.IN_Hmi_1
ellipse at (135,230)-(186,281): text "V2"; alarm colour if MAIN.fbW1210.IN_Hmi_2; taps MAIN.fbW1210.IN_Hmi_2
rectangle at (125,460)-(196,481): text "%.0f bar"; shows P1210.Bar; alarm colour if P1210.Alarm.Adver; runs INTERN ASSIGN INPUTS.PresSelCalStbd[9]:=(FALSE)
rectangle at (125,445)-(201,461): text "V%d - A P1210"; shows MAIN.fbW1210.SpdA
rectangle at (125,480)-(201,496): text "V%d - B P1211"; shows MAIN.fbW1210.SpdB
rectangle at (125,495)-(196,516): text "%.0f bar"; shows P1211.Bar; alarm colour if P1211.Alarm.Adver; runs INTERN ASSIGN INPUTS.PresSelCalStbd[9]:=(FALSE)
rectangle at (125,325)-(196,346): text "%d %%"; shows EVP1210_1 / 10; alarm colour if EVP1210_1 = 0
rectangle at (125,310)-(196,326): text "EVP1210"
rectangle at (220,55)-(291,81): text "SECONDARY / PORT"
rectangle at (710,55)-(771,81): text "PRIMARY / STBD"
rectangle at (130,55)-(191,81): text "PRIMARY / PORT"
rounded rectangle at (905,55)-(1016,96): text "CLEAR"; alarm colour if ALARMS.Clear; taps ALARMS.Clear
ellipse at (85,205)-(111,226): text "V1"; alarm colour if MAIN.fbW1208.IN_3
ellipse at (180,205)-(206,226): text "V1"; alarm colour if MAIN.fbW1210.IN_3
ellipse at (275,205)-(301,226): text "V1"; alarm colour if MAIN.fbW1212.IN_3
ellipse at (470,205)-(496,226): text "V1"; alarm colour if MAIN.fbW1206.IN_3
ellipse at (665,205)-(691,226): text "V1"; alarm colour if MAIN.fbW1604.IN_3
ellipse at (760,205)-(786,226): text "V1"; alarm colour if MAIN.fbW1202.IN_3
ellipse at (855,205)-(881,226): text "V1"; alarm colour if MAIN.fbW1602.IN_3
15 more shapes without text or variables
*)

(* Visualisation VISU_2_BOARD
rectangle at (20,550)-(331,601): text "%s"; shows INPUTS.sVisuTime
rounded rectangle at (905,505)-(1016,546): text "RETURN"; opens VISU_1_KEEL
rectangle at (15,0)-(581,51): text "DAGGERBOARD"
ellipse at (75,160)-(146,231): invisible if MAIN.fbBoard.Manual = FALSE; alarm colour if MAIN.fbBoard.MOVING_P_In
ellipse at (75,250)-(146,321): invisible if MAIN.fbBoard.Manual = FALSE; alarm colour if MAIN.fbBoard.MOVING_P_Out
ellipse at (85,170)-(136,221): text "PUMP"; invisible if MAIN.fbBoard.Manual = FALSE; alarm colour if MAIN.fbBoard.IN_Hmi_P_In; taps MAIN.fbBoard.IN_Hmi_P_In
ellipse at (85,260)-(136,311): text "EASE"; invisible if MAIN.fbBoard.Manual = FALSE; alarm colour if MAIN.fbBoard.IN_Hmi_P_Out; taps MAIN.fbBoard.IN_Hmi_P_Out
rectangle at (75,55)-(146,86): text "DGBD / PORT"
rounded rectangle at (45,95)-(116,131): text "ENABLE"; alarm colour if MAIN.aLP_Enable[11]; toggles MAIN.aLP_Enable[11]
ellipse at (195,160)-(266,231): invisible if MAIN.fbBoard.Manual = FALSE; alarm colour if MAIN.fbBoard.MOVING_S_In
ellipse at (195,250)-(266,321): invisible if MAIN.fbBoard.Manual = FALSE; alarm colour if MAIN.fbBoard.MOVING_S_Out
ellipse at (205,170)-(256,221): text "PUMP"; invisible if MAIN.fbBoard.Manual = FALSE; alarm colour if MAIN.fbBoard.IN_Hmi_S_In; taps MAIN.fbBoard.IN_Hmi_S_In
ellipse at (205,260)-(256,311): text "EASE"; invisible if MAIN.fbBoard.Manual = FALSE; alarm colour if MAIN.fbBoard.IN_Hmi_S_Out; taps MAIN.fbBoard.IN_Hmi_S_Out
rectangle at (195,55)-(266,86): text "DGBD / STBD"
rectangle at (470,300)-(571,321): text "LS801: %.1f %%"; shows LS801.Pos; alarm colour if LS801.Alarm.Adver; runs INTERN ASSIGN INPUTS.PresSelCalStbd[9]:=(FALSE)
rectangle at (0,0)-(1,1): text "{ExtendedElement},Visu\ElementDLL.ete,1,@Bargraph,121,11,3,0,1,LS801.Pos,,%,25,50,0,100,0,0,0,0,0,0,0,-13,16,700,Arial,0,255,0,255,0,0,0,0,0,0,0,0,0,,0,"
rectangle at (61,0)-(122,11): alarm colour if (LS801.Pos) < 0; left ((LS801.Pos * 1.0) - 50)  * -1.2
rectangle at (470,125)-(571,146): text "LS803: %.1f %%"; shows LS803.Pos; alarm colour if LS803.Alarm.Adver; runs INTERN ASSIGN INPUTS.PresSelCalStbd[9]:=(FALSE)
rectangle at (0,0)-(1,1): text "{ExtendedElement},Visu\ElementDLL.ete,1,@Bargraph,121,11,3,0,1,LS803.Pos,,%,25,50,0,100,0,0,0,0,0,0,0,-13,16,700,Arial,0,255,0,255,0,0,0,0,0,0,0,0,0,,0,"
rectangle at (61,0)-(122,11): alarm colour if (LS803.Pos) < 0; left ((LS803.Pos * 1.0) - 50)  * -1.2
rectangle at (520,415)-(621,436): text "P802: %.0f bar"; shows P802.Bar; alarm colour if P802.Alarm.Adver; runs INTERN ASSIGN INPUTS.PresSelCalStbd[9]:=(FALSE)
rectangle at (700,465)-(801,486): text "P1216: %.0f bar"; shows P1216.Bar; alarm colour if P1216.Alarm.Adver; runs INTERN ASSIGN INPUTS.PresSelCalStbd[9]:=(FALSE)
rectangle at (520,240)-(621,261): text "P804: %.0f bar"; shows P804.Bar; alarm colour if P804.Alarm.Adver; runs INTERN ASSIGN INPUTS.PresSelCalStbd[9]:=(FALSE)
rectangle at (700,200)-(801,221): text "P1219: %.0f bar"; shows P1219.Bar; alarm colour if P1219.Alarm.Adver; runs INTERN ASSIGN INPUTS.PresSelCalStbd[9]:=(FALSE)
ellipse at (425,300)-(466,321): text "SF801"; alarm colour if SF801.Alarm.Alarm
ellipse at (425,125)-(466,146): text "SF803"; alarm colour if SF803.Alarm.Alarm
rounded rectangle at (905,450)-(1016,491): text "CONFIG: / BOARD"; opens VISU_CFG_BOARD
rounded rectangle at (905,110)-(1016,151): text "MANUAL / BOARD"; alarm colour if MAIN.fbBoard.Manual; toggles MAIN.fbBoard.Manual
ellipse at (30,205)-(101,276): invisible if MAIN.fbBoard.Manual; alarm colour if MAIN.fbBoard.MOVING_P
ellipse at (240,205)-(311,276): invisible if MAIN.fbBoard.Manual; alarm colour if MAIN.fbBoard.MOVING_S
ellipse at (40,215)-(91,266): text "PORT"; invisible if MAIN.fbBoard.Manual; alarm colour if MAIN.fbBoard.IN_Hmi_P; taps MAIN.fbBoard.IN_Hmi_P
ellipse at (250,215)-(301,266): text "STBD"; invisible if MAIN.fbBoard.Manual; alarm colour if MAIN.fbBoard.IN_Hmi_S; taps MAIN.fbBoard.IN_Hmi_S
ellipse at (135,205)-(206,276): invisible if MAIN.fbBoard.Manual; alarm colour if MAIN.fbBoard.MOVING_C
ellipse at (145,215)-(196,266): text "CENTER"; invisible if MAIN.fbBoard.Manual; alarm colour if MAIN.fbBoard.IN_Hmi_C; taps MAIN.fbBoard.IN_Hmi_C
ellipse at (135,100)-(206,126): text "ENGINE"; alarm colour if MAIN.fbBoard.EngReady
rounded rectangle at (150,270)-(191,301): text "%d %%"; shows MAIN.fbBoard.IN_Hmi_OutPerc; invisible if MAIN.fbBoard.Manual = FALSE; editable 5..100
rounded rectangle at (150,180)-(191,211): text "%d %%"; shows MAIN.fbBoard.IN_Hmi_InPerc; invisible if MAIN.fbBoard.Manual = FALSE; editable 5..100
rectangle at (750,405)-(851,426): text "EVP1216: %d %%"; shows EVP1216_7 / 10; alarm colour if EVP1216_7 = 0
rectangle at (750,260)-(851,281): text "EVP1218: %d %%"; shows EVP1218_9 / 10; alarm colour if EVP1218_9 = 0
ellipse at (35,350)-(76,371): text "PORT"; alarm colour if MAIN.fbBoard.LS_P_Out
ellipse at (80,350)-(121,371): text "CENT"; alarm colour if MAIN.fbBoard.LS_P_Mid
ellipse at (175,350)-(216,371): text "PORT"; alarm colour if MAIN.fbBoard.LS_S_In
ellipse at (265,350)-(306,371): text "STBD"; alarm colour if MAIN.fbBoard.LS_S_Out
ellipse at (220,350)-(261,371): text "CENT"; alarm colour if MAIN.fbBoard.LS_S_Mid
rectangle at (60,455)-(141,476): text "P: %.1f %%"; shows MAIN.fbBoard.DeltaP; runs INTERN ASSIGN INPUTS.PresSelCalStbd[9]:=(FALSE)
rectangle at (60,475)-(141,496): text "S: %.1f %%"; shows MAIN.fbBoard.DeltaS; runs INTERN ASSIGN INPUTS.PresSelCalStbd[9]:=(FALSE)
rectangle at (200,455)-(281,476): text "PS: %.1f %%"; shows MAIN.fbBoard.DeltaPS; runs INTERN ASSIGN INPUTS.PresSelCalStbd[9]:=(FALSE)
rectangle at (60,440)-(141,456): text "DELTA TGT"
ellipse at (125,350)-(166,371): text "STBD"; alarm colour if MAIN.fbBoard.LS_P_In
ellipse at (255,365)-(271,381): text "S"; alarm colour if MAIN.fbBoard.LS_Safe_S_Out
ellipse at (210,365)-(226,381): text "S"; alarm colour if MAIN.fbBoard.LS_Safe_S_In
ellipse at (115,365)-(131,381): text "S"; alarm colour if MAIN.fbBoard.LS_Safe_P_In
ellipse at (70,365)-(86,381): text "S"; alarm colour if MAIN.fbBoard.LS_Safe_P_Out
ellipse at (650,395)-(701,416): text "EV802"; alarm colour if EV802
ellipse at (650,220)-(701,241): text "EV804"; alarm colour if EV804
ellipse at (650,315)-(701,336): text "EV801"; alarm colour if EV801
ellipse at (650,140)-(701,161): text "EV803"; alarm colour if EV803
rectangle at (200,440)-(281,456): text "DELTA P/S"
rounded rectangle at (225,95)-(296,131): text "FULL AUTO"; alarm colour if MAIN.aLP_Enable[12]; toggles MAIN.aLP_Enable[12]
rounded rectangle at (905,55)-(1016,96): text "CLEAR"; alarm colour if ALARMS.Clear; taps ALARMS.Clear
9 more shapes without text or variables
*)

(* Visualisation VISU_2_CAN
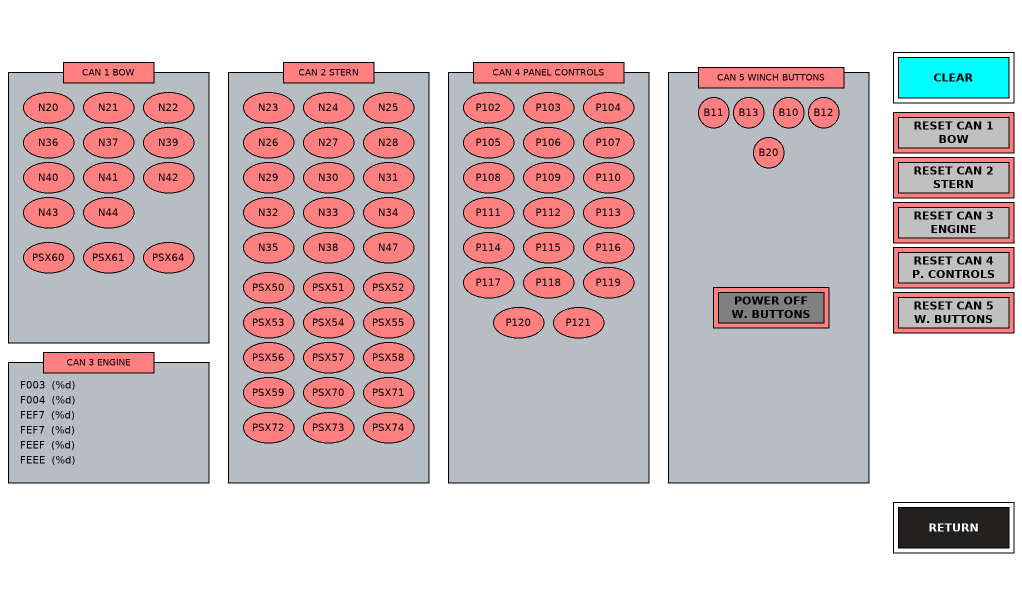
rounded rectangle at (70,60)-(161,81): text "CAN 1 BOW"; alarm colour if .CAN1_STATE = 0
rectangle at (20,0)-(331,51): text "CAN NETWORK"
rectangle at (20,550)-(331,601): text "%s"; shows INPUTS.sVisuTime
ellipse at (30,90)-(81,121): text "N20"; alarm colour if .N20_NodeState = 0
ellipse at (90,90)-(141,121): text "N21"; alarm colour if .N21_NodeState = 0
rounded rectangle at (900,500)-(1021,551): alarm colour if ALARMS.Adver
rounded rectangle at (905,505)-(1016,546): text "RETURN"; opens VISU_1_ALARMS
rounded rectangle at (290,60)-(381,81): text "CAN 2 STERN"; alarm colour if .CAN2_STATE = 0
ellipse at (150,90)-(201,121): text "N22"; alarm colour if .N22_NodeState = 0
ellipse at (310,90)-(361,121): text "N24"; alarm colour if .N24_NodeState = 0
ellipse at (250,125)-(301,156): text "N26"; alarm colour if .N26_NodeState = 0
ellipse at (250,90)-(301,121): text "N23"; alarm colour if .N23_NodeState = 0
ellipse at (370,90)-(421,121): text "N25"; alarm colour if .N25_NodeState = 0
ellipse at (310,125)-(361,156): text "N27"; alarm colour if .N27_NodeState = 0
ellipse at (30,195)-(81,226): text "N43"; alarm colour if .N43_NodeState = 0
ellipse at (90,195)-(141,226): text "N44"; alarm colour if .N44_NodeState = 0
rounded rectangle at (705,65)-(851,86): text "CAN 5 WINCH BUTTONS"; alarm colour if .CAN5_STATE = 0 OR .CAN5_STATE = 32
ellipse at (370,125)-(421,156): text "N28"; alarm colour if .N28_NodeState = 0
ellipse at (250,160)-(301,191): text "N29"; alarm colour if .N29_NodeState = 0
ellipse at (310,160)-(361,191): text "N30"; alarm colour if .N30_NodeState = 0
ellipse at (370,160)-(421,191): text "N31"; alarm colour if .N31_NodeState = 0
ellipse at (250,195)-(301,226): text "N32"; alarm colour if .N32_NodeState = 0
ellipse at (370,195)-(421,226): text "N34"; alarm colour if .N34_NodeState = 0
ellipse at (30,125)-(81,156): text "N36"; alarm colour if .N36_NodeState = 0
ellipse at (310,195)-(361,226): text "N33"; alarm colour if .N33_NodeState = 0
ellipse at (250,230)-(301,261): text "N35"; alarm colour if .N35_NodeState = 0
ellipse at (90,125)-(141,156): text "N37"; alarm colour if .N37_NodeState = 0
ellipse at (310,230)-(361,261): text "N38"; alarm colour if .N38_NodeState = 0
ellipse at (150,125)-(201,156): text "N39"; alarm colour if .N39_NodeState = 0
ellipse at (30,160)-(81,191): text "N40"; alarm colour if .N40_NodeState = 0
ellipse at (90,160)-(141,191): text "N41"; alarm colour if .N41_NodeState = 0
ellipse at (150,160)-(201,191): text "N42"; alarm colour if .N42_NodeState = 0
ellipse at (370,230)-(421,261): text "N47"; alarm colour if .N47_NodeState = 0
rounded rectangle at (480,60)-(631,81): text "CAN 4 PANEL CONTROLS"; alarm colour if .CAN4_STATE = 0
ellipse at (590,125)-(641,156): text "P107"; alarm colour if .N107_NodeState = 0
ellipse at (470,90)-(521,121): text "P102"; alarm colour if .N102_NodeState = 0
ellipse at (530,90)-(581,121): text "P103"; alarm colour if .N103_NodeState = 0
ellipse at (590,90)-(641,121): text "P104"; alarm colour if .N104_NodeState = 0
ellipse at (470,125)-(521,156): text "P105"; alarm colour if .N105_NodeState = 0
ellipse at (530,125)-(581,156): text "P106"; alarm colour if .N106_NodeState = 0
rounded rectangle at (50,350)-(161,371): text "CAN 3 ENGINE"; alarm colour if .CAN3_STATE = 0
rounded rectangle at (900,110)-(1021,151): alarm colour if .CAN1_STATE = 0
rounded rectangle at (905,115)-(1016,146): text "RESET CAN 1 / BOW"; alarm colour if OUTPUTS.ResetCan1; toggles OUTPUTS.ResetCan1
rounded rectangle at (900,155)-(1021,196): alarm colour if .CAN2_STATE = 0
rounded rectangle at (905,160)-(1016,191): text "RESET CAN 2 / STERN"; alarm colour if OUTPUTS.ResetCan2; toggles OUTPUTS.ResetCan2
rounded rectangle at (900,200)-(1021,241): alarm colour if .CAN3_STATE = 0
rounded rectangle at (905,205)-(1016,236): text "RESET CAN 3 / ENGINE"; alarm colour if OUTPUTS.ResetCan3; toggles OUTPUTS.ResetCan3
rounded rectangle at (900,290)-(1021,331): alarm colour if .CAN5_STATE = 0 OR .CAN5_STATE = 32
rounded rectangle at (905,295)-(1016,326): text "RESET CAN 5 / W. BUTTONS"; alarm colour if OUTPUTS.ResetCan5; toggles OUTPUTS.ResetCan5
rounded rectangle at (900,245)-(1021,286): alarm colour if .CAN4_STATE = 0
rounded rectangle at (905,250)-(1016,281): text "RESET CAN 4 / P. CONTROLS"; alarm colour if OUTPUTS.ResetCan4; toggles OUTPUTS.ResetCan4
ellipse at (30,240)-(81,271): text "PSX60"; alarm colour if .N60_NodeState = 0
ellipse at (90,240)-(141,271): text "PSX61"; alarm colour if .N61_NodeState = 0
ellipse at (150,240)-(201,271): text "PSX64"; alarm colour if .N64_NodeState = 0
ellipse at (250,270)-(301,301): text "PSX50"; alarm colour if .N50_NodeState = 0
ellipse at (310,270)-(361,301): text "PSX51"; alarm colour if .N51_NodeState = 0
ellipse at (370,270)-(421,301): text "PSX52"; alarm colour if .N52_NodeState = 0
ellipse at (250,305)-(301,336): text "PSX53"; alarm colour if .N53_NodeState = 0
ellipse at (310,305)-(361,336): text "PSX54"; alarm colour if .N54_NodeState = 0
ellipse at (370,305)-(421,336): text "PSX55"; alarm colour if .N55_NodeState = 0
ellipse at (250,340)-(301,371): text "PSX56"; alarm colour if .N56_NodeState = 0
ellipse at (310,340)-(361,371): text "PSX57"; alarm colour if .N57_NodeState = 0
ellipse at (370,340)-(421,371): text "PSX58"; alarm colour if .N58_NodeState = 0
ellipse at (250,375)-(301,406): text "PSX59"; alarm colour if .N59_NodeState = 0
ellipse at (310,375)-(361,406): text "PSX70"; alarm colour if .N70_NodeState = 0
ellipse at (370,375)-(421,406): text "PSX71"; alarm colour if .N71_NodeState = 0
ellipse at (250,410)-(301,441): text "PSX72"; alarm colour if .N72_NodeState = 0
ellipse at (310,410)-(361,441): text "PSX73"; alarm colour if .N73_NodeState = 0
ellipse at (370,410)-(421,441): text "PSX74"; alarm colour if .N74_NodeState = 0
rectangle at (25,375)-(106,391): text "F003	(%d)"; shows RECV_J1939.F003.Count
rectangle at (25,450)-(141,466): text "FEEE	(%d)"; shows RECV_J1939.FEEE.Count
rectangle at (25,435)-(141,451): text "FEEF	(%d)"; shows RECV_J1939.FEEF.Count
rectangle at (25,420)-(141,436): text "FEF7	(%d)"; shows RECV_J1939.FEF7.Count
rectangle at (25,405)-(141,421): text "FEF7	(%d)"; shows RECV_J1939.FEF6.Count
rectangle at (25,390)-(106,406): text "F004	(%d)"; shows RECV_J1939.F004.Count
ellipse at (590,160)-(641,191): text "P110"; alarm colour if .N110_NodeState = 0
ellipse at (470,160)-(521,191): text "P108"; alarm colour if .N108_NodeState = 0
ellipse at (530,160)-(581,191): text "P109"; alarm colour if .N109_NodeState = 0
ellipse at (590,195)-(641,226): text "P113"; alarm colour if .N113_NodeState = 0
ellipse at (470,195)-(521,226): text "P111"; alarm colour if .N111_NodeState = 0
ellipse at (530,195)-(581,226): text "P112"; alarm colour if .N112_NodeState = 0
ellipse at (590,230)-(641,261): text "P116"; alarm colour if .N116_NodeState = 0
ellipse at (470,230)-(521,261): text "P114"; alarm colour if .N114_NodeState = 0
ellipse at (530,230)-(581,261): text "P115"; alarm colour if .N115_NodeState = 0
ellipse at (590,265)-(641,296): text "P119"; alarm colour if .N119_NodeState = 0
ellipse at (470,265)-(521,296): text "P117"; alarm colour if .N117_NodeState = 0
ellipse at (530,265)-(581,296): text "P118"; alarm colour if .N118_NodeState = 0
ellipse at (780,95)-(811,126): text "B10"; alarm colour if .N10_NodeState = 0 OR .N10_NodeState = 23
ellipse at (705,95)-(736,126): text "B11"; alarm colour if .N11_NodeState = 0 OR .N11_NodeState = 23
ellipse at (815,95)-(846,126): text "B12"; alarm colour if .N12_NodeState = 0 OR .N12_NodeState = 23
ellipse at (740,95)-(771,126): text "B13"; alarm colour if .N13_NodeState = 0 OR .N13_NodeState = 23
ellipse at (760,135)-(791,166): text "B20"; alarm colour if .N20_2_NodeState = 0 OR .N20_2_NodeState = 23
rounded rectangle at (905,55)-(1016,96): text "CLEAR"; alarm colour if ALARMS.Clear; taps ALARMS.Clear
rounded rectangle at (720,285)-(836,326): alarm colour if OUTPUTS.W_CAN_PWR
rounded rectangle at (725,290)-(831,321): text "POWER OFF / W. BUTTONS"; alarm colour if OUTPUTS.W_CAN_PWR; runs INTERN ASSIGN OUTPUTS.W_CAN_CNT:=(0.0)
ellipse at (500,305)-(551,336): text "P120"; alarm colour if .N120_NodeState = 0
ellipse at (560,305)-(611,336): text "P121"; alarm colour if .N121_NodeState = 0
6 more shapes without text or variables
*)

(* Visualisation VISU_2_INPUTS
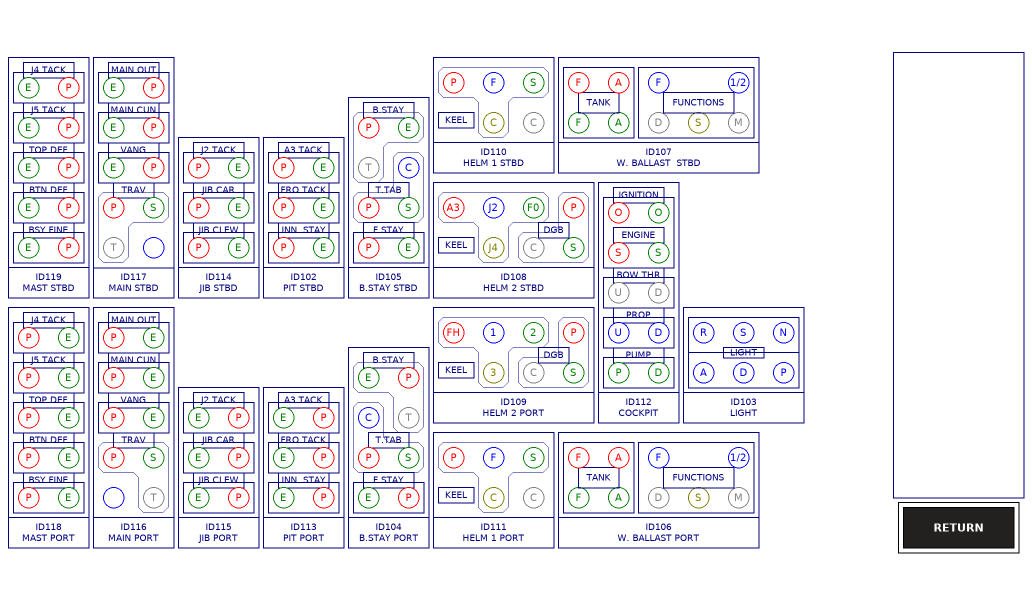
rectangle at (540,220)-(571,236): text "DGB"
rectangle at (540,345)-(571,361): text "DGB"
rectangle at (365,470)-(416,486): text "F.STAY"
rectangle at (370,430)-(411,446): text "T.TAB"
rectangle at (25,470)-(76,486): text "BSY FINE"
rectangle at (25,430)-(76,446): text "BTN DEF"
rectangle at (25,390)-(76,406): text "TOP DEF"
rectangle at (25,350)-(76,366): text "J5 TACK"
rectangle at (15,555)-(616,606): text "%s"; shows INPUTS.sVisuTime
rectangle at (20,0)-(331,51): text "INPUTS"
rectangle at (25,310)-(76,326): text "J4 TACK"
ellipse at (60,325)-(81,346): text "E"; alarm colour if .N118_IN.9
ellipse at (60,365)-(81,386): text "E"; alarm colour if .N118_IN.7
ellipse at (20,325)-(41,346): text "P"; alarm colour if .N118_IN.8
ellipse at (20,365)-(41,386): text "P"; alarm colour if .N118_IN.6
ellipse at (60,405)-(81,426): text "E"; alarm colour if .N118_IN.5
ellipse at (60,445)-(81,466): text "E"; alarm colour if .N118_IN.3
ellipse at (20,405)-(41,426): text "P"; alarm colour if .N118_IN.4
ellipse at (20,445)-(41,466): text "P"; alarm colour if .N118_IN.2
ellipse at (60,485)-(81,506): text "E"; alarm colour if .N118_IN.1
ellipse at (20,485)-(41,506): text "P"; alarm colour if .N118_IN.0
rounded rectangle at (905,505)-(1016,546): text "RETURN"; opens VISU_1_ALARMS
rectangle at (10,515)-(91,546): text "ID118 / MAST PORT"
rectangle at (10,265)-(91,296): text "ID119 / MAST STBD"
rectangle at (25,220)-(76,236): text "BSY FINE"
rectangle at (25,180)-(76,196): text "BTN DEF"
rectangle at (25,140)-(76,156): text "TOP DEF"
rectangle at (25,100)-(76,116): text "J5 TACK"
rectangle at (25,60)-(76,76): text "J4 TACK"
ellipse at (20,75)-(41,96): text "E"; alarm colour if .N119_IN.8
ellipse at (20,115)-(41,136): text "E"; alarm colour if .N119_IN.6
ellipse at (60,75)-(81,96): text "P"; alarm colour if .N119_IN.9
ellipse at (60,115)-(81,136): text "P"; alarm colour if .N119_IN.7
ellipse at (20,155)-(41,176): text "E"; alarm colour if .N119_IN.4
ellipse at (20,195)-(41,216): text "E"; alarm colour if .N119_IN.2
ellipse at (60,155)-(81,176): text "P"; alarm colour if .N119_IN.5
ellipse at (60,195)-(81,216): text "P"; alarm colour if .N119_IN.3
ellipse at (20,235)-(41,256): text "E"; alarm colour if .N119_IN.0
ellipse at (60,235)-(81,256): text "P"; alarm colour if .N119_IN.1
rectangle at (115,430)-(156,446): text "TRAV"
rectangle at (110,390)-(161,406): text "VANG"
rectangle at (110,350)-(161,366): text "MAIN CUN"
rectangle at (110,310)-(161,326): text "MAIN OUT"
ellipse at (145,325)-(166,346): text "E"; alarm colour if .N116_IN.9
ellipse at (145,365)-(166,386): text "E"; alarm colour if .N116_IN.7
ellipse at (105,325)-(126,346): text "P"; alarm colour if .N116_IN.8
ellipse at (105,365)-(126,386): text "P"; alarm colour if .N116_IN.6
ellipse at (145,405)-(166,426): text "E"; alarm colour if .N116_IN.5
ellipse at (145,445)-(166,466): text "S"; alarm colour if .N116_IN.3
ellipse at (105,405)-(126,426): text "P"; alarm colour if .N116_IN.4
ellipse at (105,445)-(126,466): text "P"; alarm colour if .N116_IN.2
ellipse at (145,485)-(166,506): text "T"; alarm colour if .N116_IN.1
ellipse at (105,485)-(126,506): alarm colour if .N116_IN.0
rectangle at (95,515)-(176,546): text "ID116 / MAIN PORT"
rectangle at (195,220)-(246,236): text "JIB CLEW"
rectangle at (195,180)-(246,196): text "JIB CAR"
rectangle at (195,140)-(246,156): text "J2 TACK"
ellipse at (230,155)-(251,176): text "E"; alarm colour if .N114_IN.5
ellipse at (230,195)-(251,216): text "E"; alarm colour if .N114_IN.3
ellipse at (190,155)-(211,176): text "P"; alarm colour if .N114_IN.4
ellipse at (190,195)-(211,216): text "P"; alarm colour if .N114_IN.2
ellipse at (230,235)-(251,256): text "E"; alarm colour if .N114_IN.1
ellipse at (190,235)-(211,256): text "P"; alarm colour if .N114_IN.0
rectangle at (180,265)-(261,296): text "ID114 / JIB STBD"
rectangle at (280,220)-(331,236): text "INN. STAY"
rectangle at (280,180)-(331,196): text "FRO TACK"
rectangle at (280,140)-(331,156): text "A3 TACK"
ellipse at (315,155)-(336,176): text "E"; alarm colour if .N102_IN.5
ellipse at (315,195)-(336,216): text "E"; alarm colour if .N102_IN.3
ellipse at (275,155)-(296,176): text "P"; alarm colour if .N102_IN.4
ellipse at (275,195)-(296,216): text "P"; alarm colour if .N102_IN.2
ellipse at (315,235)-(336,256): text "E"; alarm colour if .N102_IN.1
ellipse at (275,235)-(296,256): text "P"; alarm colour if .N102_IN.0
rectangle at (265,265)-(346,296): text "ID102 / PIT STBD"
rectangle at (435,390)-(596,421): text "ID109 / HELM 2 PORT"
ellipse at (485,485)-(506,506): text "C"; alarm colour if .N111_IN.3
ellipse at (445,445)-(466,466): text "P"; alarm colour if .N111_IN.0
rectangle at (435,515)-(556,546): text "ID111 / HELM 1 PORT"
ellipse at (525,485)-(546,506): text "C"; alarm colour if .N111_IN.5
rectangle at (350,515)-(431,546): text "ID104 / B.STAY PORT"
rectangle at (95,265)-(176,296): text "ID117 / MAIN STBD"
rectangle at (115,180)-(156,196): text "TRAV"
rectangle at (110,140)-(161,156): text "VANG"
rectangle at (110,100)-(161,116): text "MAIN CUN"
rectangle at (110,60)-(161,76): text "MAIN OUT"
ellipse at (105,75)-(126,96): text "E"; alarm colour if .N117_IN.8
ellipse at (105,115)-(126,136): text "E"; alarm colour if .N117_IN.6
ellipse at (145,75)-(166,96): text "P"; alarm colour if .N117_IN.9
ellipse at (145,115)-(166,136): text "P"; alarm colour if .N117_IN.7
ellipse at (105,155)-(126,176): text "E"; alarm colour if .N117_IN.4
ellipse at (145,195)-(166,216): text "S"; alarm colour if .N117_IN.3
ellipse at (145,155)-(166,176): text "P"; alarm colour if .N117_IN.5
ellipse at (105,195)-(126,216): text "P"; alarm colour if .N117_IN.2
ellipse at (105,235)-(126,256): text "T"; alarm colour if .N117_IN.0
ellipse at (145,235)-(166,256): alarm colour if .N117_IN.1
rectangle at (195,470)-(246,486): text "JIB CLEW"
rectangle at (195,430)-(246,446): text "JIB CAR"
rectangle at (195,390)-(246,406): text "J2 TACK"
ellipse at (190,405)-(211,426): text "E"; alarm colour if .N115_IN.4
ellipse at (190,445)-(211,466): text "E"; alarm colour if .N115_IN.2
ellipse at (230,405)-(251,426): text "P"; alarm colour if .N115_IN.5
ellipse at (230,445)-(251,466): text "P"; alarm colour if .N115_IN.3
ellipse at (190,485)-(211,506): text "E"; alarm colour if .N115_IN.0
ellipse at (230,485)-(251,506): text "P"; alarm colour if .N115_IN.1
rectangle at (180,515)-(261,546): text "ID115 / JIB PORT"
rectangle at (280,470)-(331,486): text "INN. STAY"
rectangle at (280,430)-(331,446): text "FRO TACK"
rectangle at (280,390)-(331,406): text "A3 TACK"
ellipse at (275,405)-(296,426): text "E"; alarm colour if .N113_IN.4
ellipse at (275,445)-(296,466): text "E"; alarm colour if .N113_IN.2
ellipse at (315,405)-(336,426): text "P"; alarm colour if .N113_IN.5
ellipse at (315,445)-(336,466): text "P"; alarm colour if .N113_IN.3
ellipse at (275,485)-(296,506): text "E"; alarm colour if .N113_IN.0
ellipse at (315,485)-(336,506): text "P"; alarm colour if .N113_IN.1
rectangle at (265,515)-(346,546): text "ID113 / PIT PORT"
ellipse at (360,485)-(381,506): text "E"; alarm colour if .N104_IN.0
ellipse at (400,485)-(421,506): text "P"; alarm colour if .N104_IN.1
ellipse at (400,445)-(421,466): text "S"; alarm colour if .N104_IN.3
ellipse at (360,445)-(381,466): text "P"; alarm colour if .N104_IN.2
ellipse at (360,405)-(381,426): text "C"; alarm colour if .N104_IN.4
ellipse at (400,405)-(421,426): text "T"; alarm colour if .N104_IN.5
rectangle at (365,350)-(416,366): text "B.STAY"
ellipse at (360,365)-(381,386): text "E"; alarm colour if .N104_IN.6
ellipse at (400,365)-(421,386): text "P"; alarm colour if .N104_IN.7
ellipse at (525,445)-(546,466): text "S"; alarm colour if .N111_IN.4
ellipse at (485,445)-(506,466): text "F"; alarm colour if .N111_IN.2
ellipse at (485,360)-(506,381): text "3"; alarm colour if .N109_IN.3
ellipse at (445,320)-(466,341): text "FH"; alarm colour if .N109_IN.0
ellipse at (525,360)-(546,381): text "C"; alarm colour if .N109_IN.5
ellipse at (565,360)-(586,381): text "S"; alarm colour if .N109_IN.7
ellipse at (565,320)-(586,341): text "P"; alarm colour if .N109_IN.6
ellipse at (525,320)-(546,341): text "2"; alarm colour if .N109_IN.4
ellipse at (485,320)-(506,341): text "1"; alarm colour if .N109_IN.2
ellipse at (485,110)-(506,131): text "C"; alarm colour if .N110_IN.3
ellipse at (445,70)-(466,91): text "P"; alarm colour if .N110_IN.0
rectangle at (435,140)-(556,171): text "ID110 / HELM 1 STBD"
ellipse at (525,110)-(546,131): text "C"; alarm colour if .N110_IN.5
ellipse at (525,70)-(546,91): text "S"; alarm colour if .N110_IN.4
ellipse at (485,70)-(506,91): text "F"; alarm colour if .N110_IN.2
rectangle at (435,265)-(596,296): text "ID108 / HELM 2 STBD"
ellipse at (485,235)-(506,256): text "J4"; alarm colour if .N108_IN.3
ellipse at (445,195)-(466,216): text "A3"; alarm colour if .N108_IN.0
ellipse at (525,235)-(546,256): text "C"; alarm colour if .N108_IN.5
ellipse at (565,235)-(586,256): text "S"; alarm colour if .N108_IN.7
ellipse at (565,195)-(586,216): text "P"; alarm colour if .N108_IN.6
ellipse at (525,195)-(546,216): text "F0"; alarm colour if .N108_IN.4
ellipse at (485,195)-(506,216): text "J2"; alarm colour if .N108_IN.2
rectangle at (560,140)-(761,171): text "ID107 / W. BALLAST  STBD"
rectangle at (560,515)-(761,546): text "ID106 / W. BALLAST PORT"
rectangle at (600,390)-(681,421): text "ID112 / COCKPIT"
rectangle at (685,390)-(806,421): text "ID103 / LIGHT"
rectangle at (365,220)-(416,236): text "F.STAY"
rectangle at (370,180)-(411,196): text "T.TAB"
rectangle at (350,265)-(431,296): text "ID105 / B.STAY STBD"
ellipse at (400,235)-(421,256): text "E"; alarm colour if .N105_IN.1
ellipse at (360,235)-(381,256): text "P"; alarm colour if .N105_IN.0
ellipse at (400,195)-(421,216): text "S"; alarm colour if .N105_IN.3
ellipse at (360,195)-(381,216): text "P"; alarm colour if .N105_IN.2
ellipse at (400,155)-(421,176): text "C"; alarm colour if .N105_IN.5
ellipse at (360,155)-(381,176): text "T"; alarm colour if .N105_IN.4
rectangle at (365,100)-(416,116): text "B.STAY"
ellipse at (400,115)-(421,136): text "E"; alarm colour if .N105_IN.7
ellipse at (360,115)-(381,136): text "P"; alarm colour if .N105_IN.6
rectangle at (440,485)-(476,501): text "KEEL"
rectangle at (440,360)-(476,376): text "KEEL"
rectangle at (440,235)-(476,251): text "KEEL"
rectangle at (440,110)-(476,126): text "KEEL"
ellipse at (695,360)-(716,381): text "A"; alarm colour if .N103_IN.1
ellipse at (775,320)-(796,341): text "N"; alarm colour if .N103_IN.4
ellipse at (735,360)-(756,381): text "D"; alarm colour if .N103_IN.3
ellipse at (735,320)-(756,341): text "S"; alarm colour if .N103_IN.2
ellipse at (695,320)-(716,341): text "R"; alarm colour if .N103_IN.0
ellipse at (775,360)-(796,381): text "P"; alarm colour if .N103_IN.5
rectangle at (725,345)-(766,356): text "LIGHT"
ellipse at (730,110)-(751,131): text "M"; alarm colour if .N107_IN.9
ellipse at (690,110)-(711,131): text "S"; alarm colour if .N107_IN.7
ellipse at (730,70)-(751,91): text "1/2"; alarm colour if .N107_IN.8
ellipse at (650,110)-(671,131): text "D"; alarm colour if .N107_IN.5
ellipse at (610,110)-(631,131): text "A"; alarm colour if .N107_IN.3
ellipse at (650,70)-(671,91): text "F"; alarm colour if .N107_IN.4
ellipse at (570,110)-(591,131): text "F"; alarm colour if .N107_IN.1
rectangle at (580,90)-(621,111): text "TANK"
ellipse at (570,70)-(591,91): text "F"; alarm colour if .N107_IN.0
ellipse at (610,70)-(631,91): text "A"; alarm colour if .N107_IN.2
rectangle at (665,90)-(736,111): text "FUNCTIONS"
ellipse at (730,485)-(751,506): text "M"; alarm colour if .N106_IN.9
ellipse at (690,485)-(711,506): text "S"; alarm colour if .N106_IN.7
ellipse at (730,445)-(751,466): text "1/2"; alarm colour if .N106_IN.8
ellipse at (650,485)-(671,506): text "D"; alarm colour if .N106_IN.5
ellipse at (610,485)-(631,506): text "A"; alarm colour if .N106_IN.3
ellipse at (650,445)-(671,466): text "F"; alarm colour if .N106_IN.4
ellipse at (570,485)-(591,506): text "F"; alarm colour if .N106_IN.1
rectangle at (580,465)-(621,486): text "TANK"
ellipse at (570,445)-(591,466): text "F"; alarm colour if .N106_IN.0
ellipse at (610,445)-(631,466): text "A"; alarm colour if .N106_IN.2
rectangle at (665,465)-(736,486): text "FUNCTIONS"
rectangle at (615,345)-(666,361): text "PUMP"
rectangle at (615,305)-(666,321): text "PROP"
rectangle at (615,265)-(666,281): text "BOW THR"
rectangle at (615,225)-(666,241): text "ENGINE"
rectangle at (615,185)-(666,201): text "IGNITION"
ellipse at (650,200)-(671,221): text "O"; alarm colour if .N112_IN.9
ellipse at (650,240)-(671,261): text "S"; alarm colour if .N112_IN.7
ellipse at (610,200)-(631,221): text "O"; alarm colour if .N112_IN.8
ellipse at (610,240)-(631,261): text "S"; alarm colour if .N112_IN.6
ellipse at (650,280)-(671,301): text "D"; alarm colour if .N112_IN.5
ellipse at (650,320)-(671,341): text "D"; alarm colour if .N112_IN.3
ellipse at (610,280)-(631,301): text "U"; alarm colour if .N112_IN.4
ellipse at (610,320)-(631,341): text "U"; alarm colour if .N112_IN.2
ellipse at (650,360)-(671,381): text "D"; alarm colour if .N112_IN.1
ellipse at (610,360)-(631,381): text "P"; alarm colour if .N112_IN.0
72 more shapes without text or variables
*)

(* Visualisation VISU_2_KEEL
rectangle at (20,550)-(331,601): text "%s"; shows INPUTS.sVisuTime
rounded rectangle at (905,505)-(1016,546): text "RETURN"; opens VISU_1_KEEL
rectangle at (15,0)-(581,51): text "KEEL"
rectangle at (635,175)-(736,196): text "P1001: %.0f bar"; shows P1001.Bar; alarm colour if P1001.Alarm.Adver; runs INTERN ASSIGN INPUTS.PresSelCalStbd[9]:=(FALSE)
rectangle at (475,105)-(576,126): text "LS1001: %.1f %%"; shows LS1001.Pos; alarm colour if LS1001.Alarm.Adver; runs INTERN ASSIGN INPUTS.PresSelCalStbd[9]:=(FALSE)
ellipse at (40,160)-(111,231): alarm colour if MAIN.fbKeel.MOVING_O
ellipse at (210,160)-(281,231): alarm colour if MAIN.fbKeel.MOVING_I
ellipse at (50,170)-(101,221): text "PORT"; alarm colour if MAIN.fbKeel.IN_Hmi_O; taps MAIN.fbKeel.IN_Hmi_O
ellipse at (220,170)-(271,221): text "STBD"; alarm colour if MAIN.fbKeel.IN_Hmi_I; taps MAIN.fbKeel.IN_Hmi_I
rectangle at (135,55)-(186,86): text "KEEL"
ellipse at (200,345)-(241,366): text "STBD"; alarm colour if MAIN.fbKeel.KEEL_I
ellipse at (80,345)-(121,366): text "PORT"; alarm colour if MAIN.fbKeel.KEEL_O
rounded rectangle at (40,95)-(111,131): text "ENABLE"; alarm colour if MAIN.aLP_Enable[13]; toggles MAIN.aLP_Enable[13]
rectangle at (345,175)-(446,196): text "P1002: %.0f bar"; shows P1002.Bar; alarm colour if P1002.Alarm.Adver; runs INTERN ASSIGN INPUTS.PresSelCalStbd[9]:=(FALSE)
ellipse at (140,345)-(181,366): text "CENT"; alarm colour if MAIN.fbKeel.KEEL_C
rounded rectangle at (905,110)-(1016,151): text "MANUAL / KEEL"; alarm colour if MAIN.fbKEEL.Manual; toggles MAIN.fbKEEL.Manual
ellipse at (125,160)-(196,231): alarm colour if MAIN.fbKeel.MOVING_F
ellipse at (135,170)-(186,221): text "FLOAT"; alarm colour if MAIN.fbKeel.IN_Hmi_F; taps MAIN.fbKeel.IN_Hmi_F
rounded rectangle at (905,450)-(1016,491): text "CONFIG: / KEEL"; opens VISU_CFG_KEEL
ellipse at (125,100)-(196,126): text "ENGINE"; alarm colour if MAIN.fbKEEL.EngReady
rectangle at (740,105)-(841,126): text "LS1002: %.1f %%"; shows LS1002.Pos; alarm colour if LS1002.Alarm.Adver; runs INTERN ASSIGN INPUTS.PresSelCalStbd[9]:=(FALSE)
ellipse at (760,170)-(811,191): text "SF1002"; alarm colour if SF1002.Alarm.Alarm
rectangle at (765,380)-(866,401): text "EVP1220: %d %%"; shows EVP1220_1 / 10; alarm colour if EVP1220_1 = 0
ellipse at (125,245)-(196,316): alarm colour if MAIN.fbKeel.MOVING_C
ellipse at (135,255)-(186,306): text "CENTER"; alarm colour if MAIN.fbKeel.IN_Hmi_C; taps MAIN.fbKeel.IN_Hmi_C
ellipse at (210,245)-(281,316): alarm colour if MAIN.fbKeel.MOVING_T
ellipse at (220,255)-(271,306): text "TACK"; alarm colour if MAIN.fbKeel.IN_Hmi_T; taps MAIN.fbKeel.IN_Hmi_T
ellipse at (120,345)-(141,366): text "S"; alarm colour if MAIN.fbKeel.KEEL_SO
ellipse at (180,345)-(201,366): text "S"; alarm colour if MAIN.fbKeel.KEEL_SI
rectangle at (410,505)-(516,526): text "EVP002: %d mA"; shows EVP002; alarm colour if EVP002 = 0
rectangle at (595,505)-(701,526): text "EVP001: %d mA"; shows EVP001; alarm colour if EVP001 = 0
rectangle at (630,405)-(731,426): text "EVP1005: %.0f bar"; shows EVP1005.Bar; alarm colour if EVP1005.Bar = 0
ellipse at (495,470)-(546,491): text "EV1002"; alarm colour if EV1002
ellipse at (485,400)-(536,421): text "EV1004"; alarm colour if EV1004
ellipse at (575,470)-(626,491): text "EV1001"; alarm colour if EV1001
ellipse at (565,400)-(616,421): text "EV1003"; alarm colour if EV1003
rectangle at (345,295)-(446,316): text "EVP1010: %.0f bar"; shows EVP1010.Bar; alarm colour if EVP1010.Bar = 0
ellipse at (380,400)-(431,421): text "EV1011"; alarm colour if EV1011
ellipse at (380,370)-(431,391): text "EV1012"; alarm colour if EV1012
rectangle at (305,450)-(406,471): text "P101: %.0f bar"; shows P101.Bar; alarm colour if P101.Alarm.Adver; runs INTERN ASSIGN INPUTS.PresSelCalStbd[9]:=(FALSE)
rectangle at (655,315)-(756,336): text "EVP1006: %d mA"; shows EVP1006; alarm colour if EVP1006 = 0
rectangle at (675,285)-(776,306): text "EVP1008: %d mA"; shows EVP1008; alarm colour if EVP1008 = 0
rectangle at (395,325)-(496,346): text "EVP1007: %d mA"; shows EVP1007; alarm colour if EVP1007 = 0
rectangle at (370,265)-(471,286): text "EVP1009: %d mA"; shows EVP1009; alarm colour if EVP1009 = 0
rounded rectangle at (210,95)-(281,131): text "FULL AUTO"; alarm colour if MAIN.aLP_Enable[19]; toggles MAIN.aLP_Enable[19]
rectangle at (0,0)-(1,1): text "{ExtendedElement},Visu\ElementDLL.ete,1,@Bargraph,61,11,3,0,1,LS1001.Pos,,%,25,50,50,100,0,0,0,0,0,0,0,-13,16,700,Arial,0,255,0,255,0,0,1,50,0,0,0,0,0,,0,"
rectangle at (31,0)-(62,11): alarm colour if (LS1001.Pos) > 50; left ((LS1001.Pos * 1.0) - 75)  * -1.2
rectangle at (0,0)-(1,1): text "{ExtendedElement},Visu\ElementDLL.ete,1,@Bargraph,61,11,3,0,1,LS1002.Pos,,%,25,50,50,100,0,0,0,0,0,0,0,-13,16,700,Arial,0,255,0,255,0,0,1,50,0,0,0,0,0,,0,"
rectangle at (31,0)-(62,11): alarm colour if (LS1002.Pos) > 50; left ((LS1002.Pos * 1.0) - 75)  * -1.2
rectangle at (595,525)-(701,546): text "P001: %.0f bar"; shows P001.Bar; alarm colour if P001.Alarm.Adver
rectangle at (410,525)-(516,546): text "P002: %.0f bar"; shows P002.Bar; alarm colour if P002.Alarm.Adver
ellipse at (75,435)-(126,461): text "SF1003"; alarm colour if SF1003.Alarm.Alarm
ellipse at (135,435)-(186,461): text "SF1004"; alarm colour if SF1004.Alarm.Alarm
rounded rectangle at (195,435)-(246,461): text "MUTE"; alarm colour if ALARMS.SF100x_Mute; toggles ALARMS.SF100x_Mute
rounded rectangle at (905,55)-(1016,96): text "CLEAR"; alarm colour if ALARMS.Clear; taps ALARMS.Clear
9 more shapes without text or variables
*)

